    PGN_FUEL_CELL_COMPARTMENT_INFORMATION : UDINT := UDINT#16#F349; (* < 62281 - FCCI *)
    PGN_GENSET_REAL_POWER_SETPOINT_DEMAND : UDINT := UDINT#16#F34A; (* < 62282 - GRPSD *)
    PGN_GENSET_REAL_POWER_CONTROL_2 : UDINT := UDINT#16#F34B; (* < 62283 - GRPC2 *)
    PGN_HIGH_VOLTAGE_ENERGY_STORAGE_PACK_1_DATA_12 : UDINT := UDINT#16#F34C; (* < 62284 - HVESP1D12 *)
    PGN_HIGH_VOLTAGE_ENERGY_STORAGE_PACK_1_DATA_13 : UDINT := UDINT#16#F34D; (* < 62285 - HVESP1D13 *)
    PGN_HIGH_VOLTAGE_ENERGY_STORAGE_PACK_2_DATA_12 : UDINT := UDINT#16#F34E; (* < 62286 - HVESP2D12 *)
    PGN_HIGH_VOLTAGE_ENERGY_STORAGE_PACK_2_DATA_13 : UDINT := UDINT#16#F34F; (* < 62287 - HVESP2D13 *)
    PGN_HIGH_VOLTAGE_ENERGY_STORAGE_PACK_3_DATA_12 : UDINT := UDINT#16#F350; (* < 62288 - HVESP3D12 *)
    PGN_HIGH_VOLTAGE_ENERGY_STORAGE_PACK_3_DATA_13 : UDINT := UDINT#16#F351; (* < 62289 - HVESP3D13 *)
    PGN_HIGH_VOLTAGE_ENERGY_STORAGE_PACK_4_DATA_12 : UDINT := UDINT#16#F352; (* < 62290 - HVESP4D12 *)
    PGN_HIGH_VOLTAGE_ENERGY_STORAGE_PACK_4_DATA_13 : UDINT := UDINT#16#F353; (* < 62291 - HVESP4D13 *)
    PGN_HIGH_VOLTAGE_ENERGY_STORAGE_PACK_5_DATA_12 : UDINT := UDINT#16#F354; (* < 62292 - HVESP5D12 *)
    PGN_HIGH_VOLTAGE_ENERGY_STORAGE_PACK_5_DATA_13 : UDINT := UDINT#16#F355; (* < 62293 - HVESP5D13 *)
    PGN_HIGH_VOLTAGE_ENERGY_STORAGE_PACK_6_DATA_12 : UDINT := UDINT#16#F356; (* < 62294 - HVESP6D12 *)
    PGN_HIGH_VOLTAGE_ENERGY_STORAGE_PACK_6_DATA_13 : UDINT := UDINT#16#F357; (* < 62295 - HVESP6D13 *)
    PGN_HIGH_VOLTAGE_ENERGY_STORAGE_PACK_7_DATA_12 : UDINT := UDINT#16#F358; (* < 62296 - HVESP7D12 *)
    PGN_HIGH_VOLTAGE_ENERGY_STORAGE_PACK_7_DATA_13 : UDINT := UDINT#16#F359; (* < 62297 - HVESP7D13 *)
    PGN_HIGH_VOLTAGE_ENERGY_STORAGE_PACK_8_DATA_12 : UDINT := UDINT#16#F35A; (* < 62298 - HVESP8D12 *)
    PGN_HIGH_VOLTAGE_ENERGY_STORAGE_PACK_8_DATA_13 : UDINT := UDINT#16#F35B; (* < 62299 - HVESP8D13 *)
    PGN_HIGH_VOLTAGE_ENERGY_STORAGE_PACK_9_DATA_12 : UDINT := UDINT#16#F35C; (* < 62300 - HVESP9D12 *)
    PGN_HIGH_VOLTAGE_ENERGY_STORAGE_PACK_9_DATA_13 : UDINT := UDINT#16#F35D; (* < 62301 - HVESP9D13 *)
    PGN_HIGH_VOLTAGE_ENERGY_STORAGE_PACK_10_DATA_12 : UDINT := UDINT#16#F35E; (* < 62302 - HVESP10D12 *)
    PGN_HIGH_VOLTAGE_ENERGY_STORAGE_PACK_10_DATA_13 : UDINT := UDINT#16#F35F; (* < 62303 - HVESP10D13 *)
    PGN_HIGH_VOLTAGE_ENERGY_STORAGE_PACK_11_DATA_12 : UDINT := UDINT#16#F360; (* < 62304 - HVESP11D12 *)
    PGN_HIGH_VOLTAGE_ENERGY_STORAGE_PACK_11_DATA_13 : UDINT := UDINT#16#F361; (* < 62305 - HVESP11D13 *)
    PGN_HIGH_VOLTAGE_ENERGY_STORAGE_PACK_12_DATA_12 : UDINT := UDINT#16#F362; (* < 62306 - HVESP12D12 *)
    PGN_HIGH_VOLTAGE_ENERGY_STORAGE_PACK_12_DATA_13 : UDINT := UDINT#16#F363; (* < 62307 - HVESP12D13 *)
    PGN_TRACKED_VEHICLE_DATA : UDINT := UDINT#16#F364; (* < 62308 - TVD *)
    PGN_ELECTRIFIED_ACCESSORY_PROPULSION_MOTOR_COOLANT_FAN_3_STATUS_2 : UDINT := UDINT#16#F365; (* < 62309 - EAPMCF3S2 *)
    PGN_ELECTRIFIED_ACCESSORY_PROPULSION_MOTOR_COOLANT_FAN_2_STATUS_2 : UDINT := UDINT#16#F366; (* < 62310 - EAPMCF2S2 *)
    PGN_ELECTRIFIED_ACCESSORY_PROPULSION_MOTOR_COOLANT_FAN_1_STATUS_2 : UDINT := UDINT#16#F367; (* < 62311 - EAPMCF1S2 *)
    PGN_ELECTRIFIED_ACCESSORY_POWER_ELECTRONICS_COOLANT_FAN_3_STATUS_2 : UDINT := UDINT#16#F368; (* < 62312 - EAPECF3S2 *)
    PGN_ELECTRIFIED_ACCESSORY_POWER_ELECTRONICS_COOLANT_FAN_2_STATUS_2 : UDINT := UDINT#16#F369; (* < 62313 - EAPECF2S2 *)
    PGN_ELECTRIFIED_ACCESSORY_POWER_ELECTRONICS_COOLANT_FAN_1_STATUS_2 : UDINT := UDINT#16#F36A; (* < 62314 - EAPECF1S2 *)
    PGN_ELECTRIFIED_ACCESSORY_PROPULSION_MOTOR_OIL_PUMP_STATUS_2 : UDINT := UDINT#16#F36B; (* < 62315 - EAPMOPS2 *)
    PGN_ELECTRIFIED_ACCESSORY_PROPULSION_MOTOR_COOLANT_PUMP_STATUS_2 : UDINT := UDINT#16#F36C; (* < 62316 - EAPMCPS2 *)
    PGN_ELECTRIFIED_ACCESSORY_POWER_ELECTRONICS_COOLANT_PUMP_STATUS_2 : UDINT := UDINT#16#F36D; (* < 62317 - EAPECPS2 *)
    PGN_ELECTRIFIED_ACCESSORY_GENERATOR_COOLANT_PUMP_STATUS_2 : UDINT := UDINT#16#F36E; (* < 62318 - EAGCPS2 *)
    PGN_ELECTRIFIED_ACCESSORY_GENERATOR_COOLANT_FAN_STATUS_2 : UDINT := UDINT#16#F36F; (* < 62319 - EAGCFS2 *)
    PGN_ELECTRIFIED_ACCESSORY_MOTOR_STATUS_2 : UDINT := UDINT#16#F370; (* < 62320 - EAMS2 *)
    PGN_FUEL_CELL_SYSTEM_CONTROLLER_INFORMATION : UDINT := UDINT#16#F371; (* < 62321 - FCSCI *)
    PGN_FUEL_CELL_SYSTEM_MINIMUM_POWER_INFORMATION : UDINT := UDINT#16#F372; (* < 62322 - FCSMNPI *)
    PGN_FUEL_CELL_SYSTEM_MAXIMUM_POWER_INFORMATION : UDINT := UDINT#16#F373; (* < 62323 - FCSMXPI *)
    PGN_FUEL_CELL_SYSTEM_MINIMUM_CURRENT_INFORMATION : UDINT := UDINT#16#F374; (* < 62324 - FCSMNCI *)
    PGN_FUEL_CELL_SYSTEM_MAXIMUM_CURRENT_INFORMATION : UDINT := UDINT#16#F375; (* < 62325 - FCSMXCI *)
    PGN_HYDROGEN_STORAGE_SYSTEM_INFORMATION : UDINT := UDINT#16#F376; (* < 62326 - HSSI *)
    PGN_FUEL_CELL_SYSTEM_OPERATING_STATE : UDINT := UDINT#16#F377; (* < 62327 - FCSOS *)
    PGN_FUEL_CELL_SYSTEM_OPERATIONS_REQUEST : UDINT := UDINT#16#F378; (* < 62328 - FCSOR *)
    PGN_FUEL_CELL_STACK_INFORMATION : UDINT := UDINT#16#F379; (* < 62329 - FCSI *)
    PGN_FUEL_CELL_SYSTEM_COOLANT_FAN_1_STATUS_2 : UDINT := UDINT#16#F37A; (* < 62330 - FCSCF1S2 *)
    PGN_FUEL_CELL_SYSTEM_COOLANT_FAN_2_STATUS_2 : UDINT := UDINT#16#F37B; (* < 62331 - FCSCF2S2 *)
    PGN_FUEL_CELL_SYSTEM_COOLANT_FAN_3_STATUS_2 : UDINT := UDINT#16#F37C; (* < 62332 - FCSCF3S2 *)
    PGN_FUEL_CELL_SYSTEM_COOLANT_FAN_4_STATUS_2 : UDINT := UDINT#16#F37D; (* < 62333 - FCSCF4S2 *)
    PGN_HVESS_COOLANT_PUMP_1_STATUS_2 : UDINT := UDINT#16#F37E; (* < 62334 - HVESSCP1S2 *)
    PGN_HVESS_COOLANT_PUMP_2_STATUS_2 : UDINT := UDINT#16#F37F; (* < 62335 - HVESSCP2S2 *)
    PGN_HIGH_VOLTAGE_ENERGY_STORAGE_SYSTEM_FAN_STATUS_2 : UDINT := UDINT#16#F380; (* < 62336 - HVESSFS2 *)
    PGN_PTO_DRIVE_ENGAGEMENT_2 : UDINT := UDINT#16#F381; (* < 62337 - PTODE2 *)
    PGN_FUEL_CELL_SYSTEM_HYDROGEN_PRESSURE : UDINT := UDINT#16#F382; (* < 62338 - FCSHP *)
    PGN_ENGINE_GAS_FLOW_RATE_2 : UDINT := UDINT#16#F383; (* < 62339 - EGF2 *)
    PGN_ENGINE_SUPERCHARGER_INFORMATION : UDINT := UDINT#16#F384; (* < 62340 - ESI *)
    PGN_ENGINE_DISCONNECT_CLUTCH : UDINT := UDINT#16#F385; (* < 62341 - EDC *)
    PGN_GNSS_CORRECTION_DATA : UDINT := UDINT#16#F959; (* < 63833 - GNSSCD *)
    PGN_ENGINE_CRANKCASE_VENTILATION_HEATER_INFORMATION_3 : UDINT := UDINT#16#F95A; (* < 63834 - ECVHI3 *)
    PGN_ENGINE_CRANKCASE_VENTILATION_HEATER_INFORMATION_2 : UDINT := UDINT#16#F95B; (* < 63835 - ECVHI2 *)
    PGN_ENGINE_CRANKCASE_VENTILATION_HEATER_INFORMATION_1 : UDINT := UDINT#16#F95C; (* < 63836 - ECVHI1 *)
    PGN_AIR_FUEL_RATIO_2 : UDINT := UDINT#16#F95D; (* < 63837 - AFR2 *)
    PGN_OBFCM_ENGINE_OUTPUT_ENERGY_STATIC_DATA : UDINT := UDINT#16#F95E; (* < 63838 - OBFCME *)
    PGN_OBFCM_VEHICLE_DISTANCE_STATIC_DATA : UDINT := UDINT#16#F95F; (* < 63839 - OBFCMD *)
    PGN_OBFCM_FUEL_2_STATIC_DATA : UDINT := UDINT#16#F960; (* < 63840 - OBFCMF2 *)
    PGN_OBFCM_FUEL_1_STATIC_DATA : UDINT := UDINT#16#F961; (* < 63841 - OBFCMF1 *)
    PGN_OBFCM_COUNTERS : UDINT := UDINT#16#F962; (* < 63842 - OBFCMC *)
    PGN_OBFCM_ACCUMULATORS : UDINT := UDINT#16#F963; (* < 63843 - OBFCMA *)
    PGN_OBFCM_FUEL_CONSUMPTION : UDINT := UDINT#16#F964; (* < 63844 - OBFCMFC *)
    PGN_ENGINE_VVT_SYSTEM_DATA : UDINT := UDINT#16#F965; (* < 63845 - EVVT *)
    PGN_MAINTENANCE_INFORMATION_2 : UDINT := UDINT#16#F966; (* < 63846 - MI2 *)
    PGN_ALTERNATE_FUEL_7 : UDINT := UDINT#16#F967; (* < 63847 - AF7 *)
    PGN_ENGINE_CATALYST_DIVERTER_ACTUATOR_INFORMATION : UDINT := UDINT#16#F968; (* < 63848 - ECDAI *)
    PGN_ELECTRONIC_LOGGING_DEVICE_HOURS_OF_SERVICE : UDINT := UDINT#16#F969; (* < 63849 - ELDHOS *)
    PGN_ER_DC_DC_CONVERTER_4_REFERENCES : UDINT := UDINT#16#F96A; (* < 63850 - ERDCDC4RF *)
    PGN_ER_DC_DC_CONVERTER_4_POWER_LIMITS_REQUEST : UDINT := UDINT#16#F96B; (* < 63851 - ERDCDC4PLR *)
    PGN_ER_DC_DC_CONVERTER_4_CURRENT_LIMITS_REQUEST : UDINT := UDINT#16#F96C; (* < 63852 - ERDCDC4CLR *)
    PGN_ER_DC_DC_CONVERTER_4_VOLTAGE_LIMITS_REQUEST : UDINT := UDINT#16#F96D; (* < 63853 - ERDCDC4VLR *)
    PGN_ER_DC_DC_CONVERTER_4_TEMPERATURES : UDINT := UDINT#16#F96E; (* < 63854 - ERDCDC4T *)
    PGN_ER_DC_DC_CONVERTER_4_POWER_LIMIT_SETTINGS : UDINT := UDINT#16#F96F; (* < 63855 - ERDCDC4PLS *)
    PGN_ER_DC_DC_CONVERTER_4_CURRENT_LIMITS_SETTINGS : UDINT := UDINT#16#F970; (* < 63856 - ERDCDC4CLS *)
    PGN_ER_DC_DC_CONVERTER_4_VOLTAGE_LIMIT_SETTINGS : UDINT := UDINT#16#F971; (* < 63857 - ERDCDC4VLS *)
    PGN_ER_DC_DC_CONVERTER_4_LOW_VOLTAGE : UDINT := UDINT#16#F972; (* < 63858 - ERDCDC4LV *)
    PGN_ER_DC_DC_CONVERTER_4_POWER_AND_CHASSIS_VOLTAGE : UDINT := UDINT#16#F973; (* < 63859 - ERDCDC4PCV *)
    PGN_ER_DC_DC_CONVERTER_4_VOLTAGE_AND_CURRENT : UDINT := UDINT#16#F974; (* < 63860 - ERDCDC4VC *)
    PGN_ER_DC_DC_CONVERTER_4_OPERATING_STATUS : UDINT := UDINT#16#F975; (* < 63861 - ERDCDC4OS *)
    PGN_ER_DC_DC_CONVERTER_4_CONTROL : UDINT := UDINT#16#F976; (* < 63862 - ERDCDC4C *)
    PGN_ER_DC_DC_CONVERTER_3_REFERENCES : UDINT := UDINT#16#F977; (* < 63863 - ERDCDC3RF *)
    PGN_ER_DC_DC_CONVERTER_3_POWER_LIMITS_REQUEST : UDINT := UDINT#16#F978; (* < 63864 - ERDCDC3PLR *)
    PGN_ER_DC_DC_CONVERTER_3_CURRENT_LIMITS_REQUEST : UDINT := UDINT#16#F979; (* < 63865 - ERDCDC3CLR *)
    PGN_ER_DC_DC_CONVERTER_3_VOLTAGE_LIMITS_REQUEST : UDINT := UDINT#16#F97A; (* < 63866 - ERDCDC3VLR *)
    PGN_ER_DC_DC_CONVERTER_3_TEMPERATURES : UDINT := UDINT#16#F97B; (* < 63867 - ERDCDC3T *)
    PGN_ER_DC_DC_CONVERTER_3_POWER_LIMIT_SETTINGS : UDINT := UDINT#16#F97C; (* < 63868 - ERDCDC3PLS *)
    PGN_ER_DC_DC_CONVERTER_3_CURRENT_LIMITS_SETTINGS : UDINT := UDINT#16#F97D; (* < 63869 - ERDCDC3CLS *)
    PGN_ER_DC_DC_CONVERTER_3_VOLTAGE_LIMIT_SETTINGS : UDINT := UDINT#16#F97E; (* < 63870 - ERDCDC3VLS *)
    PGN_ER_DC_DC_CONVERTER_3_LOW_VOLTAGE : UDINT := UDINT#16#F97F; (* < 63871 - ERDCDC3LV *)
    PGN_ER_DC_DC_CONVERTER_3_POWER_AND_CHASSIS_VOLTAGE : UDINT := UDINT#16#F980; (* < 63872 - ERDCDC3PCV *)
    PGN_ER_DC_DC_CONVERTER_3_VOLTAGE_AND_CURRENT : UDINT := UDINT#16#F981; (* < 63873 - ERDCDC3VC *)
    PGN_ER_DC_DC_CONVERTER_3_OPERATING_STATUS : UDINT := UDINT#16#F982; (* < 63874 - ERDCDC3OS *)
    PGN_ER_DC_DC_CONVERTER_3_CONTROL : UDINT := UDINT#16#F983; (* < 63875 - ERDCDC3C *)
    PGN_ER_DC_DC_CONVERTER_2_REFERENCES : UDINT := UDINT#16#F984; (* < 63876 - ERDCDC2RF *)
    PGN_ER_DC_DC_CONVERTER_2_POWER_LIMITS_REQUEST : UDINT := UDINT#16#F985; (* < 63877 - ERDCDC2PLR *)
    PGN_ER_DC_DC_CONVERTER_2_CURRENT_LIMITS_REQUEST : UDINT := UDINT#16#F986; (* < 63878 - ERDCDC2CLR *)
    PGN_ER_DC_DC_CONVERTER_2_VOLTAGE_LIMITS_REQUEST : UDINT := UDINT#16#F987; (* < 63879 - ERDCDC2VLR *)
    PGN_ER_DC_DC_CONVERTER_2_TEMPERATURES : UDINT := UDINT#16#F988; (* < 63880 - ERDCDC2T *)
    PGN_ER_DC_DC_CONVERTER_2_POWER_LIMIT_SETTINGS : UDINT := UDINT#16#F989; (* < 63881 - ERDCDC2PLS *)
    PGN_ER_DC_DC_CONVERTER_2_CURRENT_LIMITS_SETTINGS : UDINT := UDINT#16#F98A; (* < 63882 - ERDCDC2CLS *)
    PGN_ER_DC_DC_CONVERTER_2_VOLTAGE_LIMIT_SETTINGS : UDINT := UDINT#16#F98B; (* < 63883 - ERDCDC2VLS *)
    PGN_ER_DC_DC_CONVERTER_2_LOW_VOLTAGE : UDINT := UDINT#16#F98C; (* < 63884 - ERDCDC2LV *)
    PGN_ER_DC_DC_CONVERTER_2_POWER_AND_CHASSIS_VOLTAGE : UDINT := UDINT#16#F98D; (* < 63885 - ERDCDC2PCV *)
    PGN_ER_DC_DC_CONVERTER_2_VOLTAGE_AND_CURRENT : UDINT := UDINT#16#F98E; (* < 63886 - ERDCDC2VC *)
    PGN_ER_DC_DC_CONVERTER_2_OPERATING_STATUS : UDINT := UDINT#16#F98F; (* < 63887 - ERDCDC2OS *)
    PGN_ER_DC_DC_CONVERTER_2_CONTROL : UDINT := UDINT#16#F990; (* < 63888 - ERDCDC2C *)
    PGN_ER_DC_DC_CONVERTER_1_REFERENCES : UDINT := UDINT#16#F991; (* < 63889 - ERDCDC1RF *)
    PGN_ER_DC_DC_CONVERTER_1_POWER_LIMITS_REQUEST : UDINT := UDINT#16#F992; (* < 63890 - ERDCDC1PLR *)
    PGN_ER_DC_DC_CONVERTER_1_CURRENT_LIMITS_REQUEST : UDINT := UDINT#16#F993; (* < 63891 - ERDCDC1CLR *)
    PGN_ER_DC_DC_CONVERTER_1_VOLTAGE_LIMITS_REQUEST : UDINT := UDINT#16#F994; (* < 63892 - ERDCDC1VLR *)
    PGN_ER_DC_DC_CONVERTER_1_TEMPERATURES : UDINT := UDINT#16#F995; (* < 63893 - ERDCDC1T *)
    PGN_ER_DC_DC_CONVERTER_1_POWER_LIMIT_SETTINGS : UDINT := UDINT#16#F996; (* < 63894 - ERDCDC1PLS *)
    PGN_ER_DC_DC_CONVERTER_1_CURRENT_LIMITS_SETTINGS : UDINT := UDINT#16#F997; (* < 63895 - ERDCDC1CLS *)
    PGN_ER_DC_DC_CONVERTER_1_VOLTAGE_LIMIT_SETTINGS : UDINT := UDINT#16#F998; (* < 63896 - ERDCDC1VLS *)
    PGN_ER_DC_DC_CONVERTER_1_LOW_VOLTAGE : UDINT := UDINT#16#F999; (* < 63897 - ERDCDC1LV *)
    PGN_ER_DC_DC_CONVERTER_1_POWER_AND_CHASSIS_VOLTAGE : UDINT := UDINT#16#F99A; (* < 63898 - ERDCDC1PCV *)
    PGN_ER_DC_DC_CONVERTER_1_VOLTAGE_AND_CURRENT : UDINT := UDINT#16#F99B; (* < 63899 - ERDCDC1VC *)
    PGN_ER_DC_DC_CONVERTER_1_OPERATING_STATUS : UDINT := UDINT#16#F99C; (* < 63900 - ERDCDC1OS *)
    PGN_ER_DC_DC_CONVERTER_1_CONTROL : UDINT := UDINT#16#F99D; (* < 63901 - ERDCDC1C *)
    PGN_CAB_AIR_QUALITY_SYSTEM_INFORMATION_2 : UDINT := UDINT#16#F99E; (* < 63902 - CAQSI2 *)
    PGN_CAB_AIR_QUALITY_SYSTEM_INFORMATION_1 : UDINT := UDINT#16#F99F; (* < 63903 - CAQSI1 *)
    PGN_WELL_STIMULATION_PUMP_SYSTEM_6 : UDINT := UDINT#16#F9A0; (* < 63904 - WSP6 *)
    PGN_ENGINE_FUEL_LUBE_SYSTEMS_4 : UDINT := UDINT#16#F9A1; (* < 63905 - EFS4 *)
    PGN_ALTERNATE_FUEL_6 : UDINT := UDINT#16#F9A2; (* < 63906 - AF6 *)
    PGN_ENGINE_CATALYST_DIVERTER_ACTUATOR_CONTROL : UDINT := UDINT#16#F9A3; (* < 63907 - ECDAC *)
    PGN_AMBIENT_CONDITIONS_4 : UDINT := UDINT#16#F9A4; (* < 63908 - AMB4 *)
    PGN_ENGINE_EXHAUST_PARTICULATE_CONTROL_SYSTEM_INFO_2 : UDINT := UDINT#16#F9A5; (* < 63909 - EEPCSI2 *)
    PGN_ENGINE_EXHAUST_PARTICULATE_CONTROL_SYSTEM_INFO_1 : UDINT := UDINT#16#F9A6; (* < 63910 - EEPCSI1 *)
    PGN_AFTERTREATMENT_SYSTEM_INFORMATION_20 : UDINT := UDINT#16#F9A7; (* < 63911 - ASI20 *)
    PGN_AFTERTREATMENT_SYSTEM_INFORMATION_19 : UDINT := UDINT#16#F9A8; (* < 63912 - ASI19 *)
    PGN_AFTERTREATMENT_SYSTEM_INFORMATION_18 : UDINT := UDINT#16#F9A9; (* < 63913 - ASI18 *)
    PGN_AFTERTREATMENT_SYSTEM_INFORMATION_17 : UDINT := UDINT#16#F9AA; (* < 63914 - ASI17 *)
    PGN_AFTERTREATMENT_SYSTEM_INFORMATION_16 : UDINT := UDINT#16#F9AB; (* < 63915 - ASI16 *)
    PGN_AFTERTREATMENT_SYSTEM_INFORMATION_15 : UDINT := UDINT#16#F9AC; (* < 63916 - ASI15 *)
    PGN_AFTERTREATMENT_SYSTEM_INFORMATION_14 : UDINT := UDINT#16#F9AD; (* < 63917 - ASI14 *)
    PGN_AFTERTREATMENT_SYSTEM_INFORMATION_13 : UDINT := UDINT#16#F9AE; (* < 63918 - ASI13 *)
    PGN_AFTERTREATMENT_SYSTEM_INFORMATION_12 : UDINT := UDINT#16#F9AF; (* < 63919 - ASI12 *)
    PGN_AFTERTREATMENT_SYSTEM_INFORMATION_11 : UDINT := UDINT#16#F9B0; (* < 63920 - ASI11 *)
    PGN_AFTERTREATMENT_SYSTEM_INFORMATION_10 : UDINT := UDINT#16#F9B1; (* < 63921 - ASI10 *)
    PGN_AFTERTREATMENT_SYSTEM_INFORMATION_9 : UDINT := UDINT#16#F9B2; (* < 63922 - ASI9 *)
    PGN_ROUTE_ATTRIBUTES_PROFILE : UDINT := UDINT#16#F9B3; (* < 63923 - RTAP *)
    PGN_GENSET_SUPPORTING_FUNCTIONS_2 : UDINT := UDINT#16#F9B4; (* < 63924 - GSF2 *)
    PGN_ALTERNATOR_INFORMATION_2 : UDINT := UDINT#16#F9B5; (* < 63925 - AS2 *)
    PGN_WELL_STIMULATION_PUMP_SYSTEM_5 : UDINT := UDINT#16#F9B6; (* < 63926 - WSP5 *)
    PGN_WELL_STIMULATION_PUMP_SYSTEM_4 : UDINT := UDINT#16#F9B7; (* < 63927 - WSP4 *)
    PGN_TIRE_INFORMATION : UDINT := UDINT#16#F9B8; (* < 63928 - TI *)
    PGN_HYDROGEN_SYSTEM_STATUS : UDINT := UDINT#16#F9B9; (* < 63929 - H2SS *)
    PGN_ROUTE_WAYPOINT_GPS_COORDINATES : UDINT := UDINT#16#F9BA; (* < 63930 - RWGPSC *)
    PGN_ROUTE_INFORMATION : UDINT := UDINT#16#F9BB; (* < 63931 - RTI *)
    PGN_ENGINE_FLUID_LEVEL_PRESSURE_15 : UDINT := UDINT#16#F9BC; (* < 63932 - EFL/P15 *)
    PGN_FUEL_CELL_SYSTEM_COOLANT_INFORMATION_3 : UDINT := UDINT#16#F9BD; (* < 63933 - FCSCI3 *)
    PGN_TRANSMISSION_CONFIGURATION_3 : UDINT := UDINT#16#F9BE; (* < 63934 - TCFG3 *)
    PGN_ENRICHMENT_INFORMATION : UDINT := UDINT#16#F9BF; (* < 63935 - ENRI *)
    PGN_FUEL_CELL_SYSTEM_VOLTAGE_LIMIT_COMMAND : UDINT := UDINT#16#F9C0; (* < 63936 - FCSVLC *)
    PGN_HYDROGEN_SYSTEM_INFORMATION : UDINT := UDINT#16#F9C2; (* < 63938 - H2SYSINF *)
    PGN_AUXILIARY_INPUT_OUTPUT_STATUS_17 : UDINT := UDINT#16#F9C3; (* < 63939 - AUXIO17 *)
    PGN_AUXILIARY_INPUT_OUTPUT_STATUS_16 : UDINT := UDINT#16#F9C4; (* < 63940 - AUXIO16 *)
    PGN_AUXILIARY_INPUT_OUTPUT_STATUS_15 : UDINT := UDINT#16#F9C5; (* < 63941 - AUXIO15 *)
    PGN_AUXILIARY_INPUT_OUTPUT_STATUS_14 : UDINT := UDINT#16#F9C6; (* < 63942 - AUXIO14 *)
    PGN_AUXILIARY_INPUT_OUTPUT_STATUS_13 : UDINT := UDINT#16#F9C7; (* < 63943 - AUXIO13 *)
    PGN_AUXILIARY_INPUT_OUTPUT_STATUS_12 : UDINT := UDINT#16#F9C8; (* < 63944 - AUXIO12 *)
    PGN_AUXILIARY_INPUT_OUTPUT_STATUS_11 : UDINT := UDINT#16#F9C9; (* < 63945 - AUXIO11 *)
    PGN_AUXILIARY_INPUT_OUTPUT_STATUS_10 : UDINT := UDINT#16#F9CA; (* < 63946 - AUXIO10 *)
    PGN_AUXILIARY_INPUT_OUTPUT_STATUS_9 : UDINT := UDINT#16#F9CB; (* < 63947 - AUXIO9 *)
    PGN_AUXILIARY_INPUT_OUTPUT_STATUS_8 : UDINT := UDINT#16#F9CC; (* < 63948 - AUXIO8 *)
    PGN_AFTERTREATMENT_SYSTEM_INFORMATION_8 : UDINT := UDINT#16#F9CD; (* < 63949 - ASI8 *)
    PGN_BRAKE_TEMPERATURE_6 : UDINT := UDINT#16#F9CE; (* < 63950 - BKT6 *)
    PGN_BRAKE_TEMPERATURE_5 : UDINT := UDINT#16#F9CF; (* < 63951 - BKT5 *)
    PGN_BRAKE_TEMPERATURE_4 : UDINT := UDINT#16#F9D0; (* < 63952 - BKT4 *)
    PGN_BRAKE_TEMPERATURE_3 : UDINT := UDINT#16#F9D1; (* < 63953 - BKT3 *)
    PGN_BRAKE_TEMPERATURE_2 : UDINT := UDINT#16#F9D2; (* < 63954 - BKT2 *)
    PGN_BRAKE_TEMPERATURE_1 : UDINT := UDINT#16#F9D3; (* < 63955 - BKT1 *)
    PGN_WHEEL_BRAKE_LINING_REMAINING_INFORMATION_3 : UDINT := UDINT#16#F9D4; (* < 63956 - EBC7 *)
    PGN_WHEEL_BRAKE_LINING_REMAINING_INFORMATION_2 : UDINT := UDINT#16#F9D5; (* < 63957 - EBC6 *)
    PGN_HIGH_VOLTAGE_BUS_CONTACTOR_STATUS_3 : UDINT := UDINT#16#F9D6; (* < 63958 - HVBCS3 *)
    PGN_HIGH_VOLTAGE_BUS_CONTACTOR_STATUS_2 : UDINT := UDINT#16#F9D7; (* < 63959 - HVBCS2 *)
    PGN_HIGH_VOLTAGE_BUS_CONNECTION_COMMAND_2 : UDINT := UDINT#16#F9D8; (* < 63960 - HVBCC2 *)
    PGN_CAB_ILLUMINATION_DATA : UDINT := UDINT#16#F9D9; (* < 63961 - CID *)
    PGN_SERVICE_NEEDED_DTC_INFORMATION : UDINT := UDINT#16#F9DA; (* < 63962 - SNDI *)
    PGN_EVSE_STATUS_2 : UDINT := UDINT#16#F9DB; (* < 63963 - EVSES2 *)
    PGN_HIGH_VOLTAGE_ENERGY_STORAGE_SYSTEM_THERMAL_MANAGEMENT_SYSTEM_CHILLER_1 : UDINT := UDINT#16#F9DC; (* < 63964 - HVESSTCH1 *)
    PGN_HIGH_VOLTAGE_ENERGY_STORAGE_SYSTEM_THERMAL_MANAGEMENT_SYSTEM_CHILLER_2 : UDINT := UDINT#16#F9DD; (* < 63965 - HVESSTCH2 *)
    PGN_HIGH_VOLTAGE_ENERGY_STORAGE_SYSTEM_THERMAL_MANAGEMENT_SYSTEM_CHILLER_3 : UDINT := UDINT#16#F9DE; (* < 63966 - HVESSTCH3 *)
    PGN_HVESS_COOLANT_PUMP_1_STATUS_1 : UDINT := UDINT#16#F9DF; (* < 63967 - HVESSCP1S1 *)
    PGN_HVESS_COOLANT_PUMP_1_COMMAND : UDINT := UDINT#16#F9E0; (* < 63968 - HVESSCP1C *)
    PGN_HVESS_COOLANT_PUMP_2_STATUS_1 : UDINT := UDINT#16#F9E1; (* < 63969 - HVESSCP2S1 *)
    PGN_HVESS_COOLANT_PUMP_2_COMMAND : UDINT := UDINT#16#F9E2; (* < 63970 - HVESSCP2C *)
    PGN_HYDROGEN_SENSOR_INFORMATION : UDINT := UDINT#16#F9E3; (* < 63971 - H2SNSINF *)
    PGN_OPERATOR_INDUCEMENT_INFORMATION_2 : UDINT := UDINT#16#F9E4; (* < 63972 - OII2 *)
    PGN_OPERATOR_INDUCEMENT_VEHICLE_SPEED_INFORMATION_1 : UDINT := UDINT#16#F9E5; (* < 63973 - OIVSI1 *)
    PGN_OPERATOR_INDUCEMENT_VEHICLE_SPEED_INFORMATION_2 : UDINT := UDINT#16#F9E6; (* < 63974 - OIVSI2 *)
    PGN_ENGINE_PROTECTION_SPEED_DERATE_INFORMATION : UDINT := UDINT#16#F9E7; (* < 63975 - EPSDI *)
    PGN_ENGINE_PROTECTION_TORQUE_DERATE_INFORMATION : UDINT := UDINT#16#F9E8; (* < 63976 - EPTDI *)
    PGN_AFTERTREATMENT_SYSTEM_INFORMATION_7 : UDINT := UDINT#16#F9E9; (* < 63977 - ASI7 *)
    PGN_SAE_J2012_3_BYTE_DTC_DISPLAY : UDINT := UDINT#16#F9EA; (* < 63978 - J2012_3B *)
    PGN_HIGH_VOLTAGE_ENERGY_STORAGE_SYSTEM_INTERNAL_STATUS_5 : UDINT := UDINT#16#F9EB; (* < 63979 - HVESSIS5 *)
    PGN_HIGH_VOLTAGE_ENERGY_STORAGE_SYSTEM_INTERNAL_STATUS_6 : UDINT := UDINT#16#F9EC; (* < 63980 - HVESSIS6 *)
    PGN_HIGH_VOLTAGE_ENERGY_STORAGE_SYSTEM_INTERNAL_STATUS_7 : UDINT := UDINT#16#F9ED; (* < 63981 - HVESSIS7 *)
    PGN_ENGINE_CYLINDER_AVERAGE_IGNITION_DELAY_ANGLE_1 : UDINT := UDINT#16#F9EE; (* < 63982 - ECAIDA1 *)
    PGN_ENGINE_CYLINDER_AVERAGE_IGNITION_DELAY_ANGLE_2 : UDINT := UDINT#16#F9EF; (* < 63983 - ECAIDA2 *)
    PGN_ENGINE_CYLINDER_AVERAGE_IGNITION_DELAY_ANGLE_3 : UDINT := UDINT#16#F9F0; (* < 63984 - ECAIDA3 *)
    PGN_ENGINE_CYLINDER_AVERAGE_IGNITION_DELAY_ANGLE_4 : UDINT := UDINT#16#F9F1; (* < 63985 - ECAIDA4 *)
    PGN_ENGINE_CYLINDER_AVERAGE_IGNITION_DELAY_ANGLE_5 : UDINT := UDINT#16#F9F2; (* < 63986 - ECAIDA5 *)
    PGN_ENGINE_INDICATED_MEAN_EFFECTIVE_PRESSURE_INFORMATION_1 : UDINT := UDINT#16#F9F3; (* < 63987 - EIMEPI1 *)
    PGN_ENGINE_INDICATED_MEAN_EFFECTIVE_PRESSURE_INFORMATION_2 : UDINT := UDINT#16#F9F4; (* < 63988 - EIMEPI2 *)
    PGN_ENGINE_INDICATED_MEAN_EFFECTIVE_PRESSURE_INFORMATION_3 : UDINT := UDINT#16#F9F5; (* < 63989 - EIMEPI3 *)
    PGN_FUEL_CELL_SYSTEM_COOLANT_FAN_1_COMMAND : UDINT := UDINT#16#F9F6; (* < 63990 - FCSCF1C *)
    PGN_FUEL_CELL_SYSTEM_COOLANT_FAN_1_STATUS_1 : UDINT := UDINT#16#F9F7; (* < 63991 - FCSCF1S1 *)
    PGN_FUEL_CELL_SYSTEM_COOLANT_FAN_2_COMMAND : UDINT := UDINT#16#F9F8; (* < 63992 - FCSCF2C *)
    PGN_FUEL_CELL_SYSTEM_COOLANT_FAN_2_STATUS_1 : UDINT := UDINT#16#F9F9; (* < 63993 - FCSCF2S1 *)
    PGN_FUEL_CELL_SYSTEM_COOLANT_FAN_3_COMMAND : UDINT := UDINT#16#F9FA; (* < 63994 - FCSCF3C *)
    PGN_FUEL_CELL_SYSTEM_COOLANT_FAN_3_STATUS_1 : UDINT := UDINT#16#F9FB; (* < 63995 - FCSCF3S1 *)
    PGN_FUEL_CELL_SYSTEM_COOLANT_FAN_4_COMMAND : UDINT := UDINT#16#F9FC; (* < 63996 - FCSCF4C *)
    PGN_FUEL_CELL_SYSTEM_COOLANT_FAN_4_STATUS_1 : UDINT := UDINT#16#F9FD; (* < 63997 - FCSCF4S1 *)
    PGN_APIS_SUPPORTED : UDINT := UDINT#16#F9FE; (* < 63998 - APISUP *)
    PGN_FUEL_CELL_SYSTEM_CONFIGURATION : UDINT := UDINT#16#F9FF; (* < 63999 - FCSC *)
    PGN_FUEL_CELL_SYSTEM_COOLANT_INFORMATION_1 : UDINT := UDINT#16#FA00; (* < 64000 - FCSCI1 *)
    PGN_FUEL_CELL_SYSTEM_COOLANT_INFORMATION_2 : UDINT := UDINT#16#FA01; (* < 64001 - FCSCI2 *)
    PGN_DASH_DISPLAY_3 : UDINT := UDINT#16#FA06; (* < 64006 - DD3 *)
    PGN_VEHICLE_SPEED_PROFILE : UDINT := UDINT#16#FA07; (* < 64007 - VSP *)
    PGN_REFERENCE_TIME : UDINT := UDINT#16#FA08; (* < 64008 - REFTIME *)
    PGN_SOFTWARE_HISTORY : UDINT := UDINT#16#FA09; (* < 64009 - SH *)
    PGN_MOTOR_GENERATOR_1_THERMAL_PERFORMANCE_STATUS : UDINT := UDINT#16#FA0A; (* < 64010 - MG1TPS *)
    PGN_MOTOR_GENERATOR_2_THERMAL_PERFORMANCE_STATUS : UDINT := UDINT#16#FA0B; (* < 64011 - MG2TPS *)
    PGN_MOTOR_GENERATOR_3_THERMAL_PERFORMANCE_STATUS : UDINT := UDINT#16#FA0C; (* < 64012 - MG3TPS *)
    PGN_MOTOR_GENERATOR_4_THERMAL_PERFORMANCE_STATUS : UDINT := UDINT#16#FA0D; (* < 64013 - MG4TPS *)
    PGN_MOTOR_GENERATOR_5_THERMAL_PERFORMANCE_STATUS : UDINT := UDINT#16#FA0E; (* < 64014 - MG5TPS *)
    PGN_MOTOR_GENERATOR_6_THERMAL_PERFORMANCE_STATUS : UDINT := UDINT#16#FA0F; (* < 64015 - MG6TPS *)
    PGN_ON_BOARD_PROGRAMMING_EVENT_TIME_DATE : UDINT := UDINT#16#FA10; (* < 64016 - OBPETD *)
    PGN_AFTERTREATMENT_1_LIGHT_OFF_SCR_SERVICE_INFORMATION_1 : UDINT := UDINT#16#FA11; (* < 64017 - A1LOSCRSI1 *)
    PGN_MOTOR_GENERATOR_LOCATION_EXTENDED : UDINT := UDINT#16#FA12; (* < 64018 - MGLE *)
    PGN_COLD_START_EMISSIONS_REDUCTION_STRATEGY_CURRENT_OPERATING_CYCLE_DATA : UDINT := UDINT#16#FA13; (* < 64019 - CSERSC *)
    PGN_COLD_START_EMISSIONS_REDUCTION_STRATEGY_AVERAGE_DATA : UDINT := UDINT#16#FA14; (* < 64020 - CSERSA *)
    PGN_GENSET_SUPPORTING_FUNCTIONS : UDINT := UDINT#16#FA15; (* < 64021 - GSF *)
    PGN_HIGH_VOLTAGE_ENERGY_STORAGE_SYSTEM_INTERNAL_STATUS_1 : UDINT := UDINT#16#FA16; (* < 64022 - HVESSIS1 *)
    PGN_HIGH_VOLTAGE_ENERGY_STORAGE_SYSTEM_INTERNAL_STATUS_2 : UDINT := UDINT#16#FA17; (* < 64023 - HVESSIS2 *)
    PGN_HIGH_VOLTAGE_ENERGY_STORAGE_SYSTEM_INTERNAL_STATUS_3 : UDINT := UDINT#16#FA18; (* < 64024 - HVESSIS3 *)
    PGN_HIGH_VOLTAGE_ENERGY_STORAGE_SYSTEM_INTERNAL_STATUS_4 : UDINT := UDINT#16#FA19; (* < 64025 - HVESSIS4 *)
    PGN_ELECTRONIC_ENGINE_CONTROLLER_23 : UDINT := UDINT#16#FA1A; (* < 64026 - EEC23 *)
    PGN_ELECTRONIC_ENGINE_CONTROLLER_24 : UDINT := UDINT#16#FA1B; (* < 64027 - EEC24 *)
    PGN_ELECTRONIC_ENGINE_CONTROLLER_25 : UDINT := UDINT#16#FA1C; (* < 64028 - EEC25 *)
    PGN_HIGH_VOLTAGE_BUS_CONNECTION_COMMAND_1 : UDINT := UDINT#16#FA1D; (* < 64029 - HVBCC1 *)
    PGN_HIGH_VOLTAGE_BUS_CONTACTOR_STATUS_1 : UDINT := UDINT#16#FA1E; (* < 64030 - HVBCS1 *)
    PGN_AFTERTREATMENT_SYSTEM_INFORMATION_6 : UDINT := UDINT#16#FA1F; (* < 64031 - ASI6 *)
    PGN_EV_MULTI_CONNECTION_DC_CHARGING_LIMITS_2 : UDINT := UDINT#16#FA20; (* < 64032 - EVMCDCLIM2 *)
    PGN_EV_MULTI_CONNECTION_CHARGING_IN_PROGRESS : UDINT := UDINT#16#FA21; (* < 64033 - EVMCDCCIP *)
    PGN_SENSOR_SUPPLY_VOLTAGE : UDINT := UDINT#16#FA22; (* < 64034 - SSV *)
    PGN_MOTOR_GENERATOR_LOCATION_OBSOLETE_USE_PGN_64018 : UDINT := UDINT#16#FA23; (* < 64035 - MGL *)
    PGN_HIGH_VOLTAGE_ENERGY_STORAGE_SYSTEM_DATA_12 : UDINT := UDINT#16#FA24; (* < 64036 - HVESSD12 *)
    PGN_HIGH_VOLTAGE_ENERGY_STORAGE_SYSTEM_DATA_13 : UDINT := UDINT#16#FA25; (* < 64037 - HVESSD13 *)
    PGN_HIGH_VOLTAGE_ENERGY_STORAGE_SYSTEM_DATA_14 : UDINT := UDINT#16#FA26; (* < 64038 - HVESSD14 *)
    PGN_HIGH_VOLTAGE_ENERGY_STORAGE_PACK_1_INTERNAL_STATUS_1 : UDINT := UDINT#16#FA27; (* < 64039 - HVESP1IS1 *)
    PGN_HIGH_VOLTAGE_ENERGY_STORAGE_PACK_2_INTERNAL_STATUS_1 : UDINT := UDINT#16#FA28; (* < 64040 - HVESP2IS1 *)
    PGN_HIGH_VOLTAGE_ENERGY_STORAGE_PACK_3_INTERNAL_STATUS_1 : UDINT := UDINT#16#FA29; (* < 64041 - HVESP3IS1 *)
    PGN_HIGH_VOLTAGE_ENERGY_STORAGE_PACK_4_INTERNAL_STATUS_1 : UDINT := UDINT#16#FA2A; (* < 64042 - HVESP4IS1 *)
    PGN_HIGH_VOLTAGE_ENERGY_STORAGE_PACK_5_INTERNAL_STATUS_1 : UDINT := UDINT#16#FA2B; (* < 64043 - HVESP5IS1 *)
    PGN_HIGH_VOLTAGE_ENERGY_STORAGE_PACK_6_INTERNAL_STATUS_1 : UDINT := UDINT#16#FA2C; (* < 64044 - HVESP6IS1 *)
    PGN_HIGH_VOLTAGE_ENERGY_STORAGE_PACK_7_INTERNAL_STATUS_1 : UDINT := UDINT#16#FA2D; (* < 64045 - HVESP7IS1 *)
    PGN_HIGH_VOLTAGE_ENERGY_STORAGE_PACK_8_INTERNAL_STATUS_1 : UDINT := UDINT#16#FA2E; (* < 64046 - HVESP8IS1 *)
    PGN_HIGH_VOLTAGE_ENERGY_STORAGE_PACK_9_INTERNAL_STATUS_1 : UDINT := UDINT#16#FA2F; (* < 64047 - HVESP9IS1 *)
    PGN_HIGH_VOLTAGE_ENERGY_STORAGE_PACK_10_INTERNAL_STATUS_1 : UDINT := UDINT#16#FA30; (* < 64048 - HVESP10IS1 *)
    PGN_HIGH_VOLTAGE_ENERGY_STORAGE_PACK_11_INTERNAL_STATUS_1 : UDINT := UDINT#16#FA31; (* < 64049 - HVESP11IS1 *)
    PGN_HIGH_VOLTAGE_ENERGY_STORAGE_PACK_12_INTERNAL_STATUS_1 : UDINT := UDINT#16#FA32; (* < 64050 - HVESP12IS1 *)
    PGN_MULTI_COLOR_INDICATOR_LAMP_COMMAND : UDINT := UDINT#16#FA33; (* < 64051 - MCILC *)
    PGN_MULTI_COLOR_INDICATOR_LAMP_STATUS : UDINT := UDINT#16#FA34; (* < 64052 - MCILS *)
    PGN_REFUSE_TRUCK_BODY_INFORMATION : UDINT := UDINT#16#FA35; (* < 64053 - RTBI *)
    PGN_ENGINE_FLUID_LEVEL_PRESSURE_14 : UDINT := UDINT#16#FA36; (* < 64054 - EFL/P14 *)
    PGN_WELL_STIMULATION_TRANSMISSION_CONTROL : UDINT := UDINT#16#FA37; (* < 64055 - WSTC *)
    PGN_WELL_STIMULATION_PUMP_PROTECTION_SYSTEM_CONFIGURATION_COMMAND_1 : UDINT := UDINT#16#FA38; (* < 64056 - WSPPS1 *)
    PGN_WELL_STIMULATION_PUMP_PROTECTION_SYSTEM_CONFIGURATION_COMMAND_2 : UDINT := UDINT#16#FA39; (* < 64057 - WSPPS2 *)
    PGN_ELECTRIC_PTO_DRIVE_ENGAGEMENT_1 : UDINT := UDINT#16#FA3A; (* < 64058 - EPTODE1 *)
    PGN_ELECTRIC_PTO_1_INFORMATION : UDINT := UDINT#16#FA3B; (* < 64059 - EPTO1I *)
    PGN_ENGINE_EXHAUST_O2_SENSOR_INFORMATION : UDINT := UDINT#16#FA3C; (* < 64060 - E02SI *)
    PGN_GASEOUS_FUEL_SUPPLY_PRESSURE_3 : UDINT := UDINT#16#FA3D; (* < 64061 - GFSP3 *)
    PGN_TRAFFIC_SIGNAGE : UDINT := UDINT#16#FA3E; (* < 64062 - TS *)
    PGN_ENGINE_CONFIGURATION_4 : UDINT := UDINT#16#FA3F; (* < 64063 - EC4 *)
    PGN_ELECTRONIC_TRANSMISSION_CONTROLLER_15 : UDINT := UDINT#16#FA40; (* < 64064 - ETC15 *)
    PGN_AUTOMATED_DRIVING_SYSTEM_NETWORK_CONFIGURATION_2 : UDINT := UDINT#16#FA41; (* < 64065 - ADSNC2 *)
    PGN_AUTOMATED_DRIVING_SYSTEM_NETWORK_CONFIGURATION_1 : UDINT := UDINT#16#FA42; (* < 64066 - ADSNC1 *)
    PGN_HYBRID_OR_EV_SYSTEM_INPUTS_2 : UDINT := UDINT#16#FA43; (* < 64067 - HSI2 *)
    PGN_ENGINE_SPEED_LOAD_FACTOR_INFORMATION_2 : UDINT := UDINT#16#FA44; (* < 64068 - LF2 *)
    PGN_GENERATOR_TRIP_ENERGY_2 : UDINT := UDINT#16#FA45; (* < 64069 - GTRACE2 *)
    PGN_SECURITY_SYSTEM_MACHINE_OPERATION_INFORMATION : UDINT := UDINT#16#FA46; (* < 64070 - SSMOI *)
    PGN_ENGINE_FUEL_ACTUATOR_SERVICE_MODE : UDINT := UDINT#16#FA47; (* < 64071 - EFASM *)
    PGN_STEERING_WHEEL_CONTROLS : UDINT := UDINT#16#FA48; (* < 64072 - STWCTRL *)
    PGN_PARK_ASSIST : UDINT := UDINT#16#FA49; (* < 64073 - PA *)
    PGN_EXTENDED_DTC_INFORMATION : UDINT := UDINT#16#FA4A; (* < 64074 - DM60 *)
    PGN_AFTERTREATMENT_2_SCR_DOSING_SYSTEM_INFORMATION_5 : UDINT := UDINT#16#FA4B; (* < 64075 - A2SCRDSI5 *)
    PGN_AFTERTREATMENT_1_SCR_DOSING_SYSTEM_INFORMATION_5 : UDINT := UDINT#16#FA4C; (* < 64076 - A1SCRDSI5 *)
    PGN_EV_ECONOMY_INFORMATION : UDINT := UDINT#16#FA4D; (* < 64077 - EVEI *)
    PGN_AUTOMATED_DRIVING_SYSTEM_STATUS_2 : UDINT := UDINT#16#FA4E; (* < 64078 - ADSS2 *)
    PGN_AUTOMATED_DRIVING_SYSTEM_CONTROL_3 : UDINT := UDINT#16#FA4F; (* < 64079 - ADSC3 *)
    PGN_AFTERCOOLER_VALVE : UDINT := UDINT#16#FA50; (* < 64080 - AV *)
    PGN_ENGINE_RADIATOR_1 : UDINT := UDINT#16#FA51; (* < 64081 - ER1 *)
    PGN_ENGINE_RADIATOR_2 : UDINT := UDINT#16#FA52; (* < 64082 - ER2 *)
    PGN_GENSET_ENCLOSURE_VENTILATION : UDINT := UDINT#16#FA53; (* < 64083 - GEV *)
    PGN_HEAT_EXCHANGER_1 : UDINT := UDINT#16#FA54; (* < 64084 - HE1 *)
    PGN_HEAT_EXCHANGER_2 : UDINT := UDINT#16#FA55; (* < 64085 - HE2 *)
    PGN_HEAT_EXCHANGER_3 : UDINT := UDINT#16#FA56; (* < 64086 - HE3 *)
    PGN_HEAT_EXCHANGER_4 : UDINT := UDINT#16#FA57; (* < 64087 - HE4 *)
    PGN_ENGINE_EXHAUST_GAS_HEAT_EXCHANGER : UDINT := UDINT#16#FA58; (* < 64088 - EEGHE *)
    PGN_GENSET_ENCLOSURE_VENTILATION_LOUVER : UDINT := UDINT#16#FA59; (* < 64089 - GEVL *)
    PGN_GENSET_EXTERNAL_COOLANT_SYSTEM : UDINT := UDINT#16#FA5A; (* < 64090 - GECS *)
    PGN_EV_DC_STATUS_1 : UDINT := UDINT#16#FA5B; (* < 64091 - EVDCS1 *)
    PGN_EVSE_DC_CHARGING_LIMITS_3 : UDINT := UDINT#16#FA5C; (* < 64092 - EVSEDCLIM3 *)
    PGN_EVSE_POWER_MAX_SCHEDULE : UDINT := UDINT#16#FA5D; (* < 64093 - EVSESCHED *)
    PGN_EV_CHARGE_PROFILE : UDINT := UDINT#16#FA5E; (* < 64094 - EVCHGPROF *)
    PGN_EV_DC_CHARGING_LIMITS_2 : UDINT := UDINT#16#FA5F; (* < 64095 - EVDCLIM2 *)
    PGN_EV_DC_CHARGING_IN_PROGRESS : UDINT := UDINT#16#FA60; (* < 64096 - EVDCCIP *)
    PGN_LIGHTING_DATA_2 : UDINT := UDINT#16#FA62; (* < 64098 - LD2 *)
    PGN_LIGHTING_COMMAND_2 : UDINT := UDINT#16#FA63; (* < 64099 - LCMD2 *)
    PGN_AFTERTREATMENT_SYSTEM_INFORMATION_5 : UDINT := UDINT#16#FA64; (* < 64100 - ASI5 *)
    PGN_AFTERTREATMENT_SYSTEM_INFORMATION_4 : UDINT := UDINT#16#FA65; (* < 64101 - ASI4 *)
    PGN_AFTERTREATMENT_SYSTEM_INFORMATION_3 : UDINT := UDINT#16#FA66; (* < 64102 - ASI3 *)
    PGN_FLUID_RESISTANCE_1 : UDINT := UDINT#16#FA67; (* < 64103 - FR1 *)
    PGN_POWER_CONVERTER_2_ISOLATION_INTEGRITY_REQUEST : UDINT := UDINT#16#FA68; (* < 64104 - PC2IIR *)
    PGN_POWER_CONVERTER_1_ISOLATION_INTEGRITY_REQUEST : UDINT := UDINT#16#FA69; (* < 64105 - PC1IIR *)
    PGN_POWER_CONVERTER_2_LIMITS_REQUEST_POWER : UDINT := UDINT#16#FA6A; (* < 64106 - PC2IRP *)
    PGN_POWER_CONVERTER_2_LIMITS_REQUEST_ELECTRICAL : UDINT := UDINT#16#FA6B; (* < 64107 - PC2ILRM *)
    PGN_POWER_CONVERTER_2_LIMITS_REQUEST_DC_ENERGY_SOURCE_1 : UDINT := UDINT#16#FA6C; (* < 64108 - PC2ILRDC *)
    PGN_POWER_CONVERTER_1_LIMITS_REQUEST_DC_ENERGY_SOURCE_1 : UDINT := UDINT#16#FA6D; (* < 64109 - PC1ILRDC *)
    PGN_POWER_CONVERTER_1_LIMITS_REQUEST_ELECTRICAL : UDINT := UDINT#16#FA6E; (* < 64110 - PC1ILRM *)
    PGN_POWER_CONVERTER_1_LIMITS_REQUEST_POWER : UDINT := UDINT#16#FA6F; (* < 64111 - PC1IRP *)
    PGN_INVERTER_1_LIFETIME_DATA : UDINT := UDINT#16#FA70; (* < 64112 - PC1LD *)
    PGN_INVERTER_2_LIFETIME_DATA : UDINT := UDINT#16#FA71; (* < 64113 - PC2LD *)
    PGN_POWER_CONVERTER_2_ACTIVE_POWER_LIMITS : UDINT := UDINT#16#FA72; (* < 64114 - PC2IAPL *)
    PGN_POWER_CONVERTER_1_ACTIVE_POWER_LIMITS : UDINT := UDINT#16#FA73; (* < 64115 - PC1IAPL *)
    PGN_POWER_CONVERTER_2_REFERENCE_1 : UDINT := UDINT#16#FA74; (* < 64116 - PC2IR1 *)
    PGN_POWER_CONVERTER_2_REFERENCE_2 : UDINT := UDINT#16#FA75; (* < 64117 - PC2IR2 *)
    PGN_POWER_CONVERTER_2_TEMPERATURE : UDINT := UDINT#16#FA76; (* < 64118 - PC2IT *)
    PGN_POWER_CONVERTER_1_TEMPERATURE : UDINT := UDINT#16#FA77; (* < 64119 - PC1IT *)
    PGN_POWER_CONVERTER_1_REFERENCE_2 : UDINT := UDINT#16#FA78; (* < 64120 - PC1IR2 *)
    PGN_POWER_CONVERTER_1_REFERENCE_1 : UDINT := UDINT#16#FA79; (* < 64121 - PC1IR1 *)
    PGN_POWER_CONVERTER_1_PHASE_CURRENT : UDINT := UDINT#16#FA7A; (* < 64122 - PC1PC *)
    PGN_POWER_CONVERTER_2_PHASE_CURRENT : UDINT := UDINT#16#FA7B; (* < 64123 - S21PC *)
    PGN_POWER_CONVERTER_1_PHASE_VOLTAGE : UDINT := UDINT#16#FA7C; (* < 64124 - PC1PV *)
    PGN_POWER_CONVERTER_2_PHASE_VOLTAGE : UDINT := UDINT#16#FA7D; (* < 64125 - PC2PV *)
    PGN_POWER_CONVERTER_POWER_MODULE_SWITCH_TEMPERATURES : UDINT := UDINT#16#FA7E; (* < 64126 - SIPST *)
    PGN_POWER_CONVERTER_1_POWER_MODULE_SWITCH_POWER_SUPPLY_VOLTAGE : UDINT := UDINT#16#FA7F; (* < 64127 - PC1PSV *)
    PGN_POWER_CONVERTER_2_POWER_MODULE_SWITCH_POWER_SUPPLY_VOLTAGE : UDINT := UDINT#16#FA80; (* < 64128 - PC2PSV *)
    PGN_POWER_CONVERTER_TOTALS_1 : UDINT := UDINT#16#FA81; (* < 64129 - SIT1 *)
    PGN_TRANSFORMER_TEMPERATURES : UDINT := UDINT#16#FA82; (* < 64130 - TFMRT *)
    PGN_ELECTRIFIED_ACCESSORY_ENGINE_COOLANT_PUMP_STATUS : UDINT := UDINT#16#FA83; (* < 64131 - EAECPS *)
    PGN_HIGH_VOLTAGE_ENERGY_STORAGE_PACK_11_HISTORY : UDINT := UDINT#16#FA84; (* < 64132 - HVESP11HIST *)
    PGN_HIGH_VOLTAGE_ENERGY_STORAGE_PACK_11_CONFIGURATION : UDINT := UDINT#16#FA85; (* < 64133 - HVESP11CFG *)
    PGN_HIGH_VOLTAGE_ENERGY_STORAGE_PACK_12_HISTORY : UDINT := UDINT#16#FA86; (* < 64134 - HVESP12HIST *)
    PGN_HIGH_VOLTAGE_ENERGY_STORAGE_PACK_12_CONFIGURATION : UDINT := UDINT#16#FA87; (* < 64135 - HVESP12CFG *)
    PGN_HIGH_VOLTAGE_ENERGY_STORAGE_PACK_13_HISTORY : UDINT := UDINT#16#FA88; (* < 64136 - HVESP13HIST *)
    PGN_HIGH_VOLTAGE_ENERGY_STORAGE_PACK_13_CONFIGURATION : UDINT := UDINT#16#FA89; (* < 64137 - HVESP13CFG *)
    PGN_HIGH_VOLTAGE_ENERGY_STORAGE_PACK_14_HISTORY : UDINT := UDINT#16#FA8A; (* < 64138 - HVESP14HIST *)
    PGN_HIGH_VOLTAGE_ENERGY_STORAGE_PACK_14_CONFIGURATION : UDINT := UDINT#16#FA8B; (* < 64139 - HVESP14CFG *)
    PGN_HIGH_VOLTAGE_ENERGY_STORAGE_PACK_15_HISTORY : UDINT := UDINT#16#FA8C; (* < 64140 - HVESP15HIST *)
    PGN_HIGH_VOLTAGE_ENERGY_STORAGE_PACK_15_CONFIGURATION : UDINT := UDINT#16#FA8D; (* < 64141 - HVESP15CFG *)
    PGN_HIGH_VOLTAGE_ENERGY_STORAGE_PACK_16_HISTORY : UDINT := UDINT#16#FA8E; (* < 64142 - HVESP16HIST *)
    PGN_HIGH_VOLTAGE_ENERGY_STORAGE_PACK_16_CONFIGURATION : UDINT := UDINT#16#FA8F; (* < 64143 - HVESP16CFG *)
    PGN_HIGH_VOLTAGE_ENERGY_STORAGE_PACK_17_HISTORY : UDINT := UDINT#16#FA90; (* < 64144 - HVESP17HIST *)
    PGN_HIGH_VOLTAGE_ENERGY_STORAGE_PACK_17_CONFIGURATION : UDINT := UDINT#16#FA91; (* < 64145 - HVESP17CFG *)
    PGN_HIGH_VOLTAGE_ENERGY_STORAGE_PACK_18_HISTORY : UDINT := UDINT#16#FA92; (* < 64146 - HVESP18HIST *)
    PGN_HIGH_VOLTAGE_ENERGY_STORAGE_PACK_18_CONFIGURATION : UDINT := UDINT#16#FA93; (* < 64147 - HVESP18CFG *)
    PGN_HIGH_VOLTAGE_ENERGY_STORAGE_PACK_19_HISTORY : UDINT := UDINT#16#FA94; (* < 64148 - HVESP19HIST *)
    PGN_HIGH_VOLTAGE_ENERGY_STORAGE_PACK_19_CONFIGURATION : UDINT := UDINT#16#FA95; (* < 64149 - HVESP19CFG *)
    PGN_HIGH_VOLTAGE_ENERGY_STORAGE_PACK_20_HISTORY : UDINT := UDINT#16#FA96; (* < 64150 - HVESP20HIST *)
    PGN_HIGH_VOLTAGE_ENERGY_STORAGE_PACK_20_CONFIGURATION : UDINT := UDINT#16#FA97; (* < 64151 - HVESP20CFG *)
    PGN_HIGH_VOLTAGE_ENERGY_STORAGE_PACK_21_HISTORY : UDINT := UDINT#16#FA98; (* < 64152 - HVESP21HIST *)
    PGN_HIGH_VOLTAGE_ENERGY_STORAGE_PACK_21_CONFIGURATION : UDINT := UDINT#16#FA99; (* < 64153 - HVESP21CFG *)
    PGN_HIGH_VOLTAGE_ENERGY_STORAGE_PACK_22_HISTORY : UDINT := UDINT#16#FA9A; (* < 64154 - HVESP22HIST *)
    PGN_HIGH_VOLTAGE_ENERGY_STORAGE_PACK_22_CONFIGURATION : UDINT := UDINT#16#FA9B; (* < 64155 - HVESP22CFG *)
    PGN_HIGH_VOLTAGE_ENERGY_STORAGE_PACK_23_HISTORY : UDINT := UDINT#16#FA9C; (* < 64156 - HVESP23HIST *)
    PGN_HIGH_VOLTAGE_ENERGY_STORAGE_PACK_23_CONFIGURATION : UDINT := UDINT#16#FA9D; (* < 64157 - HVESP23CFG *)
    PGN_HIGH_VOLTAGE_ENERGY_STORAGE_PACK_24_HISTORY : UDINT := UDINT#16#FA9E; (* < 64158 - HVESP24HIST *)
    PGN_HIGH_VOLTAGE_ENERGY_STORAGE_PACK_24_CONFIGURATION : UDINT := UDINT#16#FA9F; (* < 64159 - HVESP24CFG *)
    PGN_HIGH_VOLTAGE_ENERGY_STORAGE_PACK_25_HISTORY : UDINT := UDINT#16#FAA0; (* < 64160 - HVESP25HIST *)
    PGN_HIGH_VOLTAGE_ENERGY_STORAGE_PACK_25_CONFIGURATION : UDINT := UDINT#16#FAA1; (* < 64161 - HVESP25CFG *)
    PGN_HIGH_VOLTAGE_ENERGY_STORAGE_PACK_26_HISTORY : UDINT := UDINT#16#FAA2; (* < 64162 - HVESP26HIST *)
    PGN_HIGH_VOLTAGE_ENERGY_STORAGE_PACK_26_CONFIGURATION : UDINT := UDINT#16#FAA3; (* < 64163 - HVESP26CFG *)
    PGN_AUTOMATED_DRIVING_SYSTEM_CONTROL_2 : UDINT := UDINT#16#FAA4; (* < 64164 - ADSC2 *)
    PGN_DUAL_FUEL_MODE_3 : UDINT := UDINT#16#FAA5; (* < 64165 - DFM3 *)
    PGN_DUAL_FUEL_MODE_2 : UDINT := UDINT#16#FAA6; (* < 64166 - DFM2 *)
    PGN_DUAL_FUEL_MODE_1 : UDINT := UDINT#16#FAA7; (* < 64167 - DFM1 *)
    PGN_TRANSMISSION_1_HISTORY : UDINT := UDINT#16#FAA8; (* < 64168 - T1HIST *)
    PGN_TRANSMISSION_SHAFT_TWIST_INFORMATION : UDINT := UDINT#16#FAA9; (* < 64169 - TSTI *)
    PGN_ELECTRONIC_AUXILIARY_TRANSMISSION_CONTROLLER_2 : UDINT := UDINT#16#FAAA; (* < 64170 - EATC2 *)
    PGN_HIGH_VOLTAGE_ENERGY_STORAGE_PACK_10_CONFIGURATION : UDINT := UDINT#16#FAAB; (* < 64171 - HVESP10CFG *)
    PGN_HIGH_VOLTAGE_ENERGY_STORAGE_PACK_10_HISTORY : UDINT := UDINT#16#FAAC; (* < 64172 - HVESP10HIST *)
    PGN_HIGH_VOLTAGE_ENERGY_STORAGE_PACK_9_CONFIGURATION : UDINT := UDINT#16#FAAD; (* < 64173 - HVESP9CFG *)
    PGN_HIGH_VOLTAGE_ENERGY_STORAGE_PACK_9_HISTORY : UDINT := UDINT#16#FAAE; (* < 64174 - HVESP9HIST *)
    PGN_HIGH_VOLTAGE_ENERGY_STORAGE_PACK_8_CONFIGURATION : UDINT := UDINT#16#FAAF; (* < 64175 - HVESP8CFG *)
    PGN_HIGH_VOLTAGE_ENERGY_STORAGE_PACK_8_HISTORY : UDINT := UDINT#16#FAB0; (* < 64176 - HVESP8HIST *)
    PGN_HIGH_VOLTAGE_ENERGY_STORAGE_PACK_7_CONFIGURATION : UDINT := UDINT#16#FAB1; (* < 64177 - HVESP7CFG *)
    PGN_HIGH_VOLTAGE_ENERGY_STORAGE_PACK_7_HISTORY : UDINT := UDINT#16#FAB2; (* < 64178 - HVESP7HIST *)
    PGN_AUTOSAR_TIME_SYNCHRONIZATION : UDINT := UDINT#16#FAB3; (* < 64179 - CanTSyn *)
    PGN_EV_DC_CHARGING_LIMITS_1 : UDINT := UDINT#16#FAB4; (* < 64180 - EVDCLIM1 *)
    PGN_EVSE_DC_CHARGING_LIMITS_1 : UDINT := UDINT#16#FAB5; (* < 64181 - EVSEDCLIM1 *)
    PGN_EVSE_DC_CHARGING_LIMITS_2 : UDINT := UDINT#16#FAB6; (* < 64182 - EVSEDCLIM2 *)
    PGN_EV_DC_CHARGING_TARGET : UDINT := UDINT#16#FAB7; (* < 64183 - EVDCTGT *)
    PGN_EVSE_DC_STATUS_1 : UDINT := UDINT#16#FAB8; (* < 64184 - EVSEDCS1 *)
    PGN_EVSE_1_CONTACTOR_CMD_1 : UDINT := UDINT#16#FAB9; (* < 64185 - EVSE1CC1 *)
    PGN_EVSE_1_CONTACTOR_STATUS_1 : UDINT := UDINT#16#FABA; (* < 64186 - EVSE1CS1 *)
    PGN_DIRECT_LAMP_CONTROL_COMMAND_3 : UDINT := UDINT#16#FABB; (* < 64187 - DLCC3 *)
    PGN_DIRECT_LAMP_CONTROL_DATA_3 : UDINT := UDINT#16#FABC; (* < 64188 - DLCD3 *)
    PGN_MOTOR_GENERATOR_1_LIFETIME_DATA : UDINT := UDINT#16#FABD; (* < 64189 - MG1LD *)
    PGN_MOTOR_GENERATOR_2_LIFETIME_DATA : UDINT := UDINT#16#FABE; (* < 64190 - MG2LD *)
    PGN_MOTOR_GENERATOR_3_LIFETIME_DATA : UDINT := UDINT#16#FABF; (* < 64191 - MG3LD *)
    PGN_MOTOR_GENERATOR_4_LIFETIME_DATA : UDINT := UDINT#16#FAC0; (* < 64192 - MG4LD *)
    PGN_MOTOR_GENERATOR_5_LIFETIME_DATA : UDINT := UDINT#16#FAC1; (* < 64193 - MG5LD *)
    PGN_MOTOR_GENERATOR_6_LIFETIME_DATA : UDINT := UDINT#16#FAC2; (* < 64194 - MG6LD *)
    PGN_AIR_SUPPLY_PRESSURE_3 : UDINT := UDINT#16#FAC3; (* < 64195 - AIR3 *)
    PGN_EVSE_AC_SUPPLY_VOLTAGE : UDINT := UDINT#16#FAC4; (* < 64196 - EVSEACSV *)
    PGN_EVSE_AC_3_PHASE_LOAD : UDINT := UDINT#16#FAC5; (* < 64197 - EVSEAC3PL *)
    PGN_ELECTRONIC_RETARDER_CONTROLLER_3 : UDINT := UDINT#16#FAC6; (* < 64198 - ERC3 *)
    PGN_ELECTRONIC_TRANSMISSION_CONTROLLER_14 : UDINT := UDINT#16#FAC8; (* < 64200 - ETC14 *)
    PGN_COLLISION_AVOIDANCE_SYSTEM_4 : UDINT := UDINT#16#FACB; (* < 64203 - CXD4 *)
    PGN_COLLISION_AVOIDANCE_SYSTEM_3 : UDINT := UDINT#16#FACC; (* < 64204 - CXD3 *)
    PGN_AFTERTREATMENT_1_SCR_EXHAUST_GAS_PRESSURES_2 : UDINT := UDINT#16#FACD; (* < 64205 - A1SCREGP2 *)
    PGN_PTO_INFORMATION_2 : UDINT := UDINT#16#FACE; (* < 64206 - PTO2 *)
    PGN_EVCC_DIAGNOSTIC_DATA_1 : UDINT := UDINT#16#FACF; (* < 64207 - EVCCD1 *)
    PGN_CAB_DOOR_CONTROL_2 : UDINT := UDINT#16#FAD0; (* < 64208 - CDC2 *)
    PGN_ENGINE_AVERAGE_INFORMATION_2 : UDINT := UDINT#16#FAD1; (* < 64209 - EAI2 *)
    PGN_TURBOCHARGER_INFORMATION_9 : UDINT := UDINT#16#FAD2; (* < 64210 - TCI9 *)
    PGN_AUTOMATED_DRIVING_SYSTEM_CONTROL_1 : UDINT := UDINT#16#FAD3; (* < 64211 - ADSC1 *)
    PGN_EVSE_AC_STATUS_2 : UDINT := UDINT#16#FAD4; (* < 64212 - EVSEACS2 *)
    PGN_EVSE_AC_STATUS_1 : UDINT := UDINT#16#FAD5; (* < 64213 - EVSEACS1 *)
    PGN_EVSE_STATUS_1 : UDINT := UDINT#16#FAD6; (* < 64214 - EVSES1 *)
    PGN_OBJECT_DETECTION_MESSAGE_1_1 : UDINT := UDINT#16#FAD7; (* < 64215 - ODM11 *)
    PGN_OBJECT_DETECTION_MESSAGE_2_1 : UDINT := UDINT#16#FAD8; (* < 64216 - ODM21 *)
    PGN_OBJECT_DETECTION_MESSAGE_2_2 : UDINT := UDINT#16#FAD9; (* < 64217 - ODM22 *)
    PGN_OBJECT_DETECTION_MESSAGE_2_3 : UDINT := UDINT#16#FADA; (* < 64218 - ODM23 *)
    PGN_OBJECT_DETECTION_MESSAGE_2_4 : UDINT := UDINT#16#FADB; (* < 64219 - ODM24 *)
    PGN_OBJECT_DETECTION_MESSAGE_2_5 : UDINT := UDINT#16#FADC; (* < 64220 - ODM25 *)
    PGN_OBJECT_DETECTION_MESSAGE_2_6 : UDINT := UDINT#16#FADD; (* < 64221 - ODM26 *)
    PGN_OBJECT_DETECTION_MESSAGE_2_7 : UDINT := UDINT#16#FADE; (* < 64222 - ODM27 *)
    PGN_OBJECT_DETECTION_MESSAGE_2_8 : UDINT := UDINT#16#FADF; (* < 64223 - ODM28 *)
    PGN_OBJECT_DETECTION_MESSAGE_2_9 : UDINT := UDINT#16#FAE0; (* < 64224 - ODM29 *)
    PGN_OBJECT_DETECTION_MESSAGE_2_10 : UDINT := UDINT#16#FAE1; (* < 64225 - ODM210 *)
    PGN_OBJECT_DETECTION_MESSAGE_2_11 : UDINT := UDINT#16#FAE2; (* < 64226 - ODM211 *)
    PGN_OBJECT_DETECTION_MESSAGE_2_12 : UDINT := UDINT#16#FAE3; (* < 64227 - ODM212 *)
    PGN_OBJECT_DETECTION_MESSAGE_2_13 : UDINT := UDINT#16#FAE4; (* < 64228 - ODM213 *)
    PGN_OBJECT_DETECTION_MESSAGE_2_14 : UDINT := UDINT#16#FAE5; (* < 64229 - ODM214 *)
    PGN_OBJECT_DETECTION_MESSAGE_2_15 : UDINT := UDINT#16#FAE6; (* < 64230 - ODM215 *)
    PGN_OBJECT_DETECTION_MESSAGE_2_16 : UDINT := UDINT#16#FAE7; (* < 64231 - ODM216 *)
    PGN_OBJECT_DETECTION_MESSAGE_2_17 : UDINT := UDINT#16#FAE8; (* < 64232 - ODM217 *)
    PGN_OBJECT_DETECTION_MESSAGE_2_18 : UDINT := UDINT#16#FAE9; (* < 64233 - ODM218 *)
    PGN_OBJECT_DETECTION_MESSAGE_2_19 : UDINT := UDINT#16#FAEA; (* < 64234 - ODM219 *)
    PGN_OBJECT_DETECTION_MESSAGE_2_20 : UDINT := UDINT#16#FAEB; (* < 64235 - ODM220 *)
    PGN_OBJECT_DETECTION_MESSAGE_2_21 : UDINT := UDINT#16#FAEC; (* < 64236 - ODM221 *)
    PGN_TEMPERATURE_SENSING_MODULE_1 : UDINT := UDINT#16#FAED; (* < 64237 - TSM1 *)
    PGN_TEMPERATURE_SENSING_MODULE_2 : UDINT := UDINT#16#FAEE; (* < 64238 - TSM2 *)
    PGN_AFTERTREATMENT_2_SCR_SERVICE_INFORMATION_3 : UDINT := UDINT#16#FAEF; (* < 64239 - A2SCRSI3 *)
    PGN_AFTERTREATMENT_1_SCR_SERVICE_INFORMATION_3 : UDINT := UDINT#16#FAF0; (* < 64240 - A1SCRSI3 *)
    PGN_PSA_TIMES_LIFETIME_HOURS : UDINT := UDINT#16#FAF1; (* < 64241 - PSATL *)
    PGN_PSA_TIMES_STORED_100_HOURS : UDINT := UDINT#16#FAF2; (* < 64242 - PSATS *)
    PGN_PSA_TIMES_ACTIVE_100_HOURS : UDINT := UDINT#16#FAF3; (* < 64243 - PSATA *)
    PGN_HYBRID_CHARGE_DEPLETING_OR_INCREASING_OPERATION_LIFETIME_HOURS : UDINT := UDINT#16#FAF4; (* < 64244 - HCDIOL *)
    PGN_HYBRID_CHARGE_DEPLETING_OR_INCREASING_OPERATION_STORED_100_HOURS : UDINT := UDINT#16#FAF5; (* < 64245 - HCDIOS *)
    PGN_HYBRID_CHARGE_DEPLETING_OR_INCREASING_OPERATION_ACTIVE_100_HOURS : UDINT := UDINT#16#FAF6; (* < 64246 - HCDIOA *)
    PGN_AFTERTREATMENT_1_HISTORICAL_INFORMATION_3 : UDINT := UDINT#16#FAF7; (* < 64247 - AT1HI3 *)
    PGN_ENGINE_MAXIMUM_NET_TORQUE_MAP : UDINT := UDINT#16#FAF8; (* < 64248 - ENGMXT *)
    PGN_AFTERTREATMENT_1_SCR_2_NOX_MASS_AND_NH3_STORAGE : UDINT := UDINT#16#FAF9; (* < 64249 - ATNXMS2 *)
    PGN_AFTERTREATMENT_1_SCR_1_NOX_MASS_AND_NH3_STORAGE : UDINT := UDINT#16#FAFA; (* < 64250 - ATNXMS1 *)
    PGN_EVAPORATIVE_SYSTEM_PRESSURE_AND_CONTROL : UDINT := UDINT#16#FAFB; (* < 64251 - ESPC *)
    PGN_GHG_TRACKING_LIFETIME_ARRAY_DATA : UDINT := UDINT#16#FAFC; (* < 64252 - GHGTL *)
    PGN_GHG_TRACKING_STORED_100_HOUR_ARRAY_DATA : UDINT := UDINT#16#FAFD; (* < 64253 - GHGTS *)
    PGN_GHG_TRACKING_ACTIVE_100_HOUR_ARRAY_DATA : UDINT := UDINT#16#FAFE; (* < 64254 - GHGTA *)
    PGN_GREEN_HOUSE_GAS_STORED_100_HOUR_ACTIVE_TECHNOLOGY_TRACKING : UDINT := UDINT#16#FAFF; (* < 64255 - GHGTTS *)
    PGN_GREEN_HOUSE_GAS_ACTIVE_100_HOUR_ACTIVE_TECHNOLOGY_TRACKING : UDINT := UDINT#16#FB00; (* < 64256 - GHGTTA *)
    PGN_GREEN_HOUSE_GAS_LIFETIME_ACTIVE_TECHNOLOGY_TRACKING : UDINT := UDINT#16#FB01; (* < 64257 - GHGTTL *)
    PGN_NOX_TRACKING_ENGINE_ACTIVITY_LIFETIME_FUEL_CONSUMPTION_BINS : UDINT := UDINT#16#FB02; (* < 64258 - NTFCEA *)
    PGN_NOX_TRACKING_ENGINE_ACTIVITY_LIFETIME_ENGINE_RUN_TIME_BINS : UDINT := UDINT#16#FB03; (* < 64259 - NTEHEA *)
    PGN_NOX_TRACKING_ENGINE_ACTIVITY_LIFETIME_VEHICLE_DISTANCE_BINS : UDINT := UDINT#16#FB04; (* < 64260 - NTVMEA *)
    PGN_NOX_TRACKING_ENGINE_ACTIVITY_LIFETIME_ENGINE_OUTPUT_ENERGY_BINS : UDINT := UDINT#16#FB05; (* < 64261 - NTEEEA *)
    PGN_NOX_TRACKING_VALID_NOX_LIFETIME_FUEL_CONSUMPTION_BINS : UDINT := UDINT#16#FB06; (* < 64262 - NTFCV *)
    PGN_NOX_TRACKING_VALID_NOX_LIFETIME_ENGINE_RUN_TIME_BINS : UDINT := UDINT#16#FB07; (* < 64263 - NTEHV *)
    PGN_NOX_TRACKING_VALID_NOX_LIFETIME_VEHICLE_DISTANCE_BINS : UDINT := UDINT#16#FB08; (* < 64264 - NTVMV *)
    PGN_NOX_TRACKING_VALID_NOX_LIFETIME_ENGINE_OUTPUT_ENERGY_BINS : UDINT := UDINT#16#FB09; (* < 64265 - NTEEV *)
    PGN_NOX_TRACKING_VALID_NOX_LIFETIME_ENGINE_OUT_NOX_MASS_BINS : UDINT := UDINT#16#FB0A; (* < 64266 - NTENV *)
    PGN_NOX_TRACKING_VALID_NOX_LIFETIME_SYSTEM_OUT_NOX_MASS_BINS : UDINT := UDINT#16#FB0B; (* < 64267 - NTSNV *)
    PGN_NOX_TRACKING_STORED_100_HOUR_FUEL_CONSUMPTION_BINS : UDINT := UDINT#16#FB0C; (* < 64268 - NTFCS *)
    PGN_NOX_TRACKING_STORED_100_HOUR_ENGINE_RUN_TIME_BINS : UDINT := UDINT#16#FB0D; (* < 64269 - NTEHS *)
    PGN_NOX_TRACKING_STORED_100_HOUR_VEHICLE_DISTANCE_BINS : UDINT := UDINT#16#FB0E; (* < 64270 - NTVMS *)
    PGN_NOX_TRACKING_STORED_100_HOUR_ENGINE_OUTPUT_ENERGY_BINS : UDINT := UDINT#16#FB0F; (* < 64271 - NTEES *)
    PGN_NOX_TRACKING_STORED_100_HOUR_ENGINE_OUT_NOX_MASS_BINS : UDINT := UDINT#16#FB10; (* < 64272 - NTENS *)
    PGN_NOX_TRACKING_STORED_100_HOUR_SYSTEM_OUT_NOX_MASS_BINS : UDINT := UDINT#16#FB11; (* < 64273 - NTSNS *)
    PGN_NOX_TRACKING_ACTIVE_100_HOUR_FUEL_CONSUMPTION_BINS : UDINT := UDINT#16#FB12; (* < 64274 - NTFCA *)
    PGN_NOX_TRACKING_ACTIVE_100_HOUR_ENGINE_RUN_TIME_BINS : UDINT := UDINT#16#FB13; (* < 64275 - NTEHA *)
    PGN_NOX_TRACKING_ACTIVE_100_HOUR_VEHICLE_DISTANCE_BINS : UDINT := UDINT#16#FB14; (* < 64276 - NTVMA *)
    PGN_NOX_TRACKING_ACTIVE_100_HOUR_ENGINE_OUTPUT_ENERGY_BINS : UDINT := UDINT#16#FB15; (* < 64277 - NTEEA *)
    PGN_NOX_TRACKING_ACTIVE_100_HOUR_ENGINE_OUT_NOX_MASS_BINS : UDINT := UDINT#16#FB16; (* < 64278 - NTENA *)
    PGN_NOX_TRACKING_ACTIVE_100_HOUR_SYSTEM_OUT_NOX_MASS_BINS : UDINT := UDINT#16#FB17; (* < 64279 - NTSNA *)
    PGN_MOTOR_GENERATOR_6_INVERTER_CONTROL_2 : UDINT := UDINT#16#FB18; (* < 64280 - MG6IC2 *)
    PGN_MOTOR_GENERATOR_6_INVERTER_LIMITS_REQUEST_POWER : UDINT := UDINT#16#FB19; (* < 64281 - MG6IRP *)
    PGN_MOTOR_GENERATOR_6_INVERTER_LIMITS_REQUEST_MECHANICAL : UDINT := UDINT#16#FB1A; (* < 64282 - MG6ILRM *)
    PGN_MOTOR_GENERATOR_6_INVERTER_LIMITS_REQUEST_DC_SIDE : UDINT := UDINT#16#FB1B; (* < 64283 - MG6ILRDC *)
    PGN_MOTOR_GENERATOR_6_INVERTER_ISOLATION_INTEGRITY_REQUEST : UDINT := UDINT#16#FB1C; (* < 64284 - MG6IIR *)
    PGN_MOTOR_GENERATOR_5_INVERTER_CONTROL_2 : UDINT := UDINT#16#FB1D; (* < 64285 - MG5IC2 *)
    PGN_MOTOR_GENERATOR_5_INVERTER_LIMITS_REQUEST_POWER : UDINT := UDINT#16#FB1E; (* < 64286 - MG5IRP *)
    PGN_MOTOR_GENERATOR_5_INVERTER_LIMITS_REQUEST_MECHANICAL : UDINT := UDINT#16#FB1F; (* < 64287 - MG5ILRM *)
    PGN_MOTOR_GENERATOR_5_INVERTER_LIMITS_REQUEST_DC_SIDE : UDINT := UDINT#16#FB20; (* < 64288 - MG5ILRDC *)
    PGN_MOTOR_GENERATOR_5_INVERTER_ISOLATION_INTEGRITY_REQUEST : UDINT := UDINT#16#FB21; (* < 64289 - MG5IIR *)
    PGN_MOTOR_GENERATOR_4_INVERTER_CONTROL_2 : UDINT := UDINT#16#FB22; (* < 64290 - MG4IC2 *)
    PGN_MOTOR_GENERATOR_4_INVERTER_LIMITS_REQUEST_POWER : UDINT := UDINT#16#FB23; (* < 64291 - MG4IRP *)
    PGN_MOTOR_GENERATOR_4_INVERTER_LIMITS_REQUEST_MECHANICAL : UDINT := UDINT#16#FB24; (* < 64292 - MG4ILRM *)
    PGN_MOTOR_GENERATOR_4_INVERTER_LIMITS_REQUEST_DC_SIDE : UDINT := UDINT#16#FB25; (* < 64293 - MG4ILRDC *)
    PGN_MOTOR_GENERATOR_4_INVERTER_ISOLATION_INTEGRITY_REQUEST : UDINT := UDINT#16#FB26; (* < 64294 - MG4IIR *)
    PGN_MOTOR_GENERATOR_3_INVERTER_CONTROL_2 : UDINT := UDINT#16#FB27; (* < 64295 - MG3IC2 *)
    PGN_MOTOR_GENERATOR_3_INVERTER_LIMITS_REQUEST_POWER : UDINT := UDINT#16#FB28; (* < 64296 - MG3IRP *)
    PGN_MOTOR_GENERATOR_3_INVERTER_LIMITS_REQUEST_MECHANICAL : UDINT := UDINT#16#FB29; (* < 64297 - MG3ILRM *)
    PGN_MOTOR_GENERATOR_3_INVERTER_LIMITS_REQUEST_DC_SIDE : UDINT := UDINT#16#FB2A; (* < 64298 - MG3ILRDC *)
    PGN_MOTOR_GENERATOR_3_INVERTER_ISOLATION_INTEGRITY_REQUEST : UDINT := UDINT#16#FB2B; (* < 64299 - MG3IIR *)
    PGN_DIAGNOSTIC_READINESS_4 : UDINT := UDINT#16#FB2C; (* < 64300 - DM59 *)
    PGN_TURBOCHARGER_INFORMATION_8 : UDINT := UDINT#16#FB2D; (* < 64301 - TCI8 *)
    PGN_WINCH_INFORMATION_2 : UDINT := UDINT#16#FB2E; (* < 64302 - WINCH2 *)
    PGN_MOTOR_GENERATOR_6_INVERTER_REFERENCE_1 : UDINT := UDINT#16#FB2F; (* < 64303 - MG6IR1 *)
    PGN_MOTOR_GENERATOR_6_INVERTER_STATUS_1 : UDINT := UDINT#16#FB30; (* < 64304 - MG6IS1 *)
    PGN_MOTOR_GENERATOR_6_INVERTER_REFERENCE_2 : UDINT := UDINT#16#FB31; (* < 64305 - MG6IR2 *)
    PGN_MOTOR_GENERATOR_6_INVERTER_TEMPERATURE : UDINT := UDINT#16#FB32; (* < 64306 - MG6IT *)
    PGN_MOTOR_GENERATOR_6_INVERTER_MOTOR_TEMPERATURE : UDINT := UDINT#16#FB33; (* < 64307 - MG6IMT *)
    PGN_MOTOR_GENERATOR_6_INVERTER_ISOLATION_INTEGRITY : UDINT := UDINT#16#FB34; (* < 64308 - MG6II *)
    PGN_MOTOR_GENERATOR_6_INVERTER_ACTIVE_POWER_LIMITS : UDINT := UDINT#16#FB35; (* < 64309 - MG6IAPL *)
    PGN_MOTOR_GENERATOR_5_INVERTER_REFERENCE_1 : UDINT := UDINT#16#FB36; (* < 64310 - MG5IR1 *)
    PGN_MOTOR_GENERATOR_5_INVERTER_STATUS_1 : UDINT := UDINT#16#FB37; (* < 64311 - MG5IS1 *)
    PGN_MOTOR_GENERATOR_5_INVERTER_REFERENCE_2 : UDINT := UDINT#16#FB38; (* < 64312 - MG5IR2 *)
    PGN_MOTOR_GENERATOR_5_INVERTER_TEMPERATURE : UDINT := UDINT#16#FB39; (* < 64313 - MG5IT *)
    PGN_MOTOR_GENERATOR_5_INVERTER_MOTOR_TEMPERATURE : UDINT := UDINT#16#FB3A; (* < 64314 - MG5IMT *)
    PGN_MOTOR_GENERATOR_5_INVERTER_ISOLATION_INTEGRITY : UDINT := UDINT#16#FB3B; (* < 64315 - MG5II *)
    PGN_MOTOR_GENERATOR_5_INVERTER_ACTIVE_POWER_LIMITS : UDINT := UDINT#16#FB3C; (* < 64316 - MG5IAPL *)
    PGN_MOTOR_GENERATOR_4_INVERTER_REFERENCE_1 : UDINT := UDINT#16#FB3D; (* < 64317 - MG4IR1 *)
    PGN_MOTOR_GENERATOR_4_INVERTER_STATUS_1 : UDINT := UDINT#16#FB3E; (* < 64318 - MG4IS1 *)
    PGN_MOTOR_GENERATOR_4_INVERTER_REFERENCE_2 : UDINT := UDINT#16#FB3F; (* < 64319 - MG4IR2 *)
    PGN_MOTOR_GENERATOR_4_INVERTER_TEMPERATURE : UDINT := UDINT#16#FB40; (* < 64320 - MG4IT *)
    PGN_MOTOR_GENERATOR_4_INVERTER_MOTOR_TEMPERATURE : UDINT := UDINT#16#FB41; (* < 64321 - MG4IMT *)
    PGN_MOTOR_GENERATOR_4_INVERTER_ISOLATION_INTEGRITY : UDINT := UDINT#16#FB42; (* < 64322 - MG4II *)
    PGN_MOTOR_GENERATOR_4_INVERTER_ACTIVE_POWER_LIMITS : UDINT := UDINT#16#FB43; (* < 64323 - MG4IAPL *)
    PGN_MOTOR_GENERATOR_3_INVERTER_REFERENCE_1 : UDINT := UDINT#16#FB44; (* < 64324 - MG3IR1 *)
    PGN_MOTOR_GENERATOR_3_INVERTER_STATUS_1 : UDINT := UDINT#16#FB45; (* < 64325 - MG3IS1 *)
    PGN_MOTOR_GENERATOR_3_INVERTER_REFERENCE_2 : UDINT := UDINT#16#FB46; (* < 64326 - MG3IR2 *)
    PGN_MOTOR_GENERATOR_3_INVERTER_TEMPERATURE : UDINT := UDINT#16#FB47; (* < 64327 - MG3IT *)
    PGN_MOTOR_GENERATOR_3_INVERTER_MOTOR_TEMPERATURE : UDINT := UDINT#16#FB48; (* < 64328 - MG3IMT *)
    PGN_MOTOR_GENERATOR_3_INVERTER_ISOLATION_INTEGRITY : UDINT := UDINT#16#FB49; (* < 64329 - MG3II *)
    PGN_MOTOR_GENERATOR_3_INVERTER_ACTIVE_POWER_LIMITS : UDINT := UDINT#16#FB4A; (* < 64330 - MG3IAPL *)
    PGN_AUTOMATED_DRIVING_SYSTEM_STATUS_1 : UDINT := UDINT#16#FB4B; (* < 64331 - ADSS1 *)
    PGN_CAB_CLIMATE_SYSTEM_INFORMATION_2 : UDINT := UDINT#16#FB4C; (* < 64332 - CCSI2 *)
    PGN_MAINTENANCE_INFORMATION_1 : UDINT := UDINT#16#FB4D; (* < 64333 - MI1 *)
    PGN_HOIST_CONTROL_INFORMATION : UDINT := UDINT#16#FB4E; (* < 64334 - HCI1 *)
    PGN_HIGH_VOLTAGE_ENERGY_STORAGE_PACK_6_HISTORY : UDINT := UDINT#16#FB4F; (* < 64335 - HVESP6HIST *)
    PGN_HIGH_VOLTAGE_ENERGY_STORAGE_PACK_6_CONFIGURATION : UDINT := UDINT#16#FB50; (* < 64336 - HVESP6CFG *)
    PGN_HIGH_VOLTAGE_ENERGY_STORAGE_PACK_5_HISTORY : UDINT := UDINT#16#FB51; (* < 64337 - HVESP5HIST *)
    PGN_HIGH_VOLTAGE_ENERGY_STORAGE_PACK_5_CONFIGURATION : UDINT := UDINT#16#FB52; (* < 64338 - HVESP5CFG *)
    PGN_HIGH_VOLTAGE_ENERGY_STORAGE_PACK_4_HISTORY : UDINT := UDINT#16#FB53; (* < 64339 - HVESP4HIST *)
    PGN_HIGH_VOLTAGE_ENERGY_STORAGE_PACK_4_CONFIGURATION : UDINT := UDINT#16#FB54; (* < 64340 - HVESP4CFG *)
    PGN_HIGH_VOLTAGE_ENERGY_STORAGE_PACK_3_HISTORY : UDINT := UDINT#16#FB55; (* < 64341 - HVESP3HIST *)
    PGN_HIGH_VOLTAGE_ENERGY_STORAGE_PACK_3_CONFIGURATION : UDINT := UDINT#16#FB56; (* < 64342 - HVESP3CFG *)
    PGN_HIGH_VOLTAGE_ENERGY_STORAGE_PACK_2_HISTORY : UDINT := UDINT#16#FB57; (* < 64343 - HVESP2HIST *)
    PGN_HIGH_VOLTAGE_ENERGY_STORAGE_PACK_2_CONFIGURATION : UDINT := UDINT#16#FB58; (* < 64344 - HVESP2CFG *)
    PGN_HIGH_VOLTAGE_ENERGY_STORAGE_PACK_1_HISTORY : UDINT := UDINT#16#FB59; (* < 64345 - HVESP1HIST *)
    PGN_HIGH_VOLTAGE_ENERGY_STORAGE_PACK_1_CONFIGURATION : UDINT := UDINT#16#FB5A; (* < 64346 - HVESP1CFG *)
    PGN_VEHICLE_FIRE_SUPPRESSION_SYSTEM_MODULE_1_DETECTOR_DATA : UDINT := UDINT#16#FB5B; (* < 64347 - VFSSM1DET *)
    PGN_VEHICLE_FIRE_SUPPRESSION_SYSTEM_MODULE_2_DETECTOR_DATA : UDINT := UDINT#16#FB5C; (* < 64348 - VFSSM2DET *)
    PGN_VEHICLE_FIRE_SUPPRESSION_SYSTEM_MODULE_3_DETECTOR_DATA : UDINT := UDINT#16#FB5D; (* < 64349 - VFSSM3DET *)
    PGN_VEHICLE_FIRE_SUPPRESSION_SYSTEM_MODULE_4_DETECTOR_DATA : UDINT := UDINT#16#FB5E; (* < 64350 - VFSSM4DET *)
    PGN_VEHICLE_FIRE_SUPPRESSION_SYSTEM_MODULE_1_AUXILIARY_DATA : UDINT := UDINT#16#FB5F; (* < 64351 - VFSSM1AUX *)
    PGN_VEHICLE_FIRE_SUPPRESSION_SYSTEM_MODULE_2_AUXILIARY_DATA : UDINT := UDINT#16#FB60; (* < 64352 - VFSSM2AUX *)
    PGN_VEHICLE_FIRE_SUPPRESSION_SYSTEM_MODULE_3_AUXILIARY_DATA : UDINT := UDINT#16#FB61; (* < 64353 - VFSSM3AUX *)
    PGN_VEHICLE_FIRE_SUPPRESSION_SYSTEM_MODULE_4_AUXILIARY_DATA : UDINT := UDINT#16#FB62; (* < 64354 - VFSSM4AUX *)
    PGN_VEHICLE_FIRE_SUPPRESSION_SYSTEM_MODULE_1_NAMES : UDINT := UDINT#16#FB63; (* < 64355 - VFSSM1NAMES *)
    PGN_VEHICLE_FIRE_SUPPRESSION_SYSTEM_MODULE_2_NAMES : UDINT := UDINT#16#FB64; (* < 64356 - VFSSM2NAMES *)
    PGN_VEHICLE_FIRE_SUPPRESSION_SYSTEM_MODULE_3_NAMES : UDINT := UDINT#16#FB65; (* < 64357 - VFSSM3NAMES *)
    PGN_VEHICLE_FIRE_SUPPRESSION_SYSTEM_MODULE_4_NAMES : UDINT := UDINT#16#FB66; (* < 64358 - VFSSM4NAMES *)
    PGN_MOTOR_GENERATOR_2_INVERTER_ACTIVE_POWER_LIMITS : UDINT := UDINT#16#FB67; (* < 64359 - MG2IAPL *)
    PGN_MOTOR_GENERATOR_2_INVERTER_ISOLATION_INTEGRITY : UDINT := UDINT#16#FB68; (* < 64360 - MG2II *)
    PGN_MOTOR_GENERATOR_1_INVERTER_ACTIVE_POWER_LIMITS : UDINT := UDINT#16#FB69; (* < 64361 - MG1IAPL *)
    PGN_MOTOR_GENERATOR_1_INVERTER_ISOLATION_INTEGRITY : UDINT := UDINT#16#FB6A; (* < 64362 - MG1II *)
    PGN_HIGH_VOLTAGE_BUS_INFORMATION : UDINT := UDINT#16#FB6B; (* < 64363 - HVBI *)
    PGN_MOTOR_GENERATOR_2_INVERTER_REFERENCE_1 : UDINT := UDINT#16#FB6C; (* < 64364 - MG2IR1 *)
    PGN_MOTOR_GENERATOR_2_INVERTER_STATUS_1 : UDINT := UDINT#16#FB6D; (* < 64365 - MG2IS1 *)
    PGN_MOTOR_GENERATOR_2_INVERTER_REFERENCE_2 : UDINT := UDINT#16#FB6E; (* < 64366 - MG2IR2 *)
    PGN_MOTOR_GENERATOR_2_INVERTER_TEMPERATURE : UDINT := UDINT#16#FB6F; (* < 64367 - MG2IT *)
    PGN_MOTOR_GENERATOR_2_INVERTER_MOTOR_TEMPERATURE : UDINT := UDINT#16#FB70; (* < 64368 - MG2IMT *)
    PGN_MOTOR_GENERATOR_1_INVERTER_MOTOR_TEMPERATURE : UDINT := UDINT#16#FB71; (* < 64369 - MG1IMT *)
    PGN_MOTOR_GENERATOR_1_INVERTER_TEMPERATURE : UDINT := UDINT#16#FB72; (* < 64370 - MG1IT *)
    PGN_MOTOR_GENERATOR_1_INVERTER_REFERENCE_2 : UDINT := UDINT#16#FB73; (* < 64371 - MG1IR2 *)
    PGN_MOTOR_GENERATOR_1_INVERTER_STATUS_1 : UDINT := UDINT#16#FB74; (* < 64372 - MG1IS1 *)
    PGN_MOTOR_GENERATOR_1_INVERTER_REFERENCE_1 : UDINT := UDINT#16#FB75; (* < 64373 - MG1IR1 *)
    PGN_PERSONNEL_DETECT_STATUS : UDINT := UDINT#16#FB76; (* < 64374 - PDS *)
    PGN_ENGINE_CYLINDER_PRESSURE_GAMMA_1 : UDINT := UDINT#16#FB77; (* < 64375 - ECPG1 *)
    PGN_ENGINE_CYLINDER_PRESSURE_GAMMA_2 : UDINT := UDINT#16#FB78; (* < 64376 - ECPG2 *)
    PGN_ENGINE_CYLINDER_PRESSURE_GAMMA_3 : UDINT := UDINT#16#FB79; (* < 64377 - ECPG3 *)
    PGN_ENGINE_CYLINDER_PRESSURE_GAMMA_4 : UDINT := UDINT#16#FB7A; (* < 64378 - ECPG4 *)
    PGN_ENGINE_CYLINDER_PRESSURE_GAMMA_5 : UDINT := UDINT#16#FB7B; (* < 64379 - ECPG5 *)
    PGN_WAKE_UP_AND_SLEEP : UDINT := UDINT#16#FB7C; (* < 64380 - WAKE *)
    PGN_ELECTRIFIED_ACCESSORY_GENERATOR_COOLANT_PUMP_STATUS_1 : UDINT := UDINT#16#FB7D; (* < 64381 - EAGCPS1 *)
    PGN_ELECTRIFIED_ACCESSORY_GENERATOR_COOLANT_FAN_STATUS_1 : UDINT := UDINT#16#FB7E; (* < 64382 - EAGCFS1 *)
    PGN_WELL_STIMULATION_PUMP_SYSTEM_FILTER_INFORMATION : UDINT := UDINT#16#FB7F; (* < 64383 - WSPF *)
    PGN_PTO_GOVERNOR_CONFIGURATION : UDINT := UDINT#16#FB80; (* < 64384 - PTOGC *)
    PGN_ON_BOARD_PROGRAMMING_2 : UDINT := UDINT#16#FB81; (* < 64385 - OBP2 *)
    PGN_PRIMARY_OR_REAR_HITCH_YAW : UDINT := UDINT#16#FB82; (* < 64386 - RHY *)
    PGN_SECONDARY_OR_FRONT_HITCH_YAW : UDINT := UDINT#16#FB83; (* < 64387 - FHY *)
    PGN_OPERATOR_STATUS : UDINT := UDINT#16#FB84; (* < 64388 - OPSTAT *)
    PGN_ENGINE_IDLE_MANAGEMENT_INFORMATION : UDINT := UDINT#16#FB85; (* < 64389 - EIMI *)
    PGN_ALCOHOL_INTERLOCK_TO_VEHICLE : UDINT := UDINT#16#FB86; (* < 64390 - AITOV *)
    PGN_VEHICLE_TO_ALCOHOL_INTERLOCK : UDINT := UDINT#16#FB87; (* < 64391 - VTOAI *)
    PGN_MARINE_CONTROL_INFORMATION_3 : UDINT := UDINT#16#FB88; (* < 64392 - MCI3 *)
    PGN_ENGINE_FLUID_LEVEL_PRESSURE_13 : UDINT := UDINT#16#FB89; (* < 64393 - EFL/P13 *)
    PGN_HIGH_VOLTAGE_ENERGY_STORAGE_SYSTEM_DATA_11 : UDINT := UDINT#16#FB8A; (* < 64394 - HVESSD11 *)
    PGN_ECONOMY_MODE_INACTIVE_HOURS : UDINT := UDINT#16#FB8B; (* < 64395 - EMIH *)
    PGN_ECONOMY_MODE_ESTIMATED_INSTANTANEOUS_FUEL_SAVINGS_RATE : UDINT := UDINT#16#FB8C; (* < 64396 - EMEIFSR *)
    PGN_ECONOMY_MODE_ACTIVE_HOURS : UDINT := UDINT#16#FB8D; (* < 64397 - EMAH *)
    PGN_ECONOMY_MODE_FUEL_USED : UDINT := UDINT#16#FB8E; (* < 64398 - EMFU *)
    PGN_ECONOMY_MODE_ESTIMATED_FUEL_SAVINGS : UDINT := UDINT#16#FB8F; (* < 64399 - EMEFS *)
    PGN_DC_DC_CONVERTER_4_VOLTAGE : UDINT := UDINT#16#FB90; (* < 64400 - DCDC4V *)
    PGN_DC_DC_CONVERTER_3_VOLTAGE : UDINT := UDINT#16#FB91; (* < 64401 - DCDC3V *)
    PGN_DC_DC_CONVERTER_2_VOLTAGE : UDINT := UDINT#16#FB92; (* < 64402 - DCDC2V *)
    PGN_DC_DC_CONVERTER_1_VOLTAGE : UDINT := UDINT#16#FB93; (* < 64403 - DCDC1V *)
    PGN_ELECTRONIC_ENGINE_CONTROLLER_22 : UDINT := UDINT#16#FB94; (* < 64404 - EEC22 *)
    PGN_ENGINE_HOURS_2 : UDINT := UDINT#16#FB95; (* < 64405 - HOURS2 *)
    PGN_ENGINE_INFORMATION_3 : UDINT := UDINT#16#FB96; (* < 64406 - EI3 *)
    PGN_VEHICLE_ELECTRICAL_POWER_15 : UDINT := UDINT#16#FB97; (* < 64407 - VEP15 *)
    PGN_EXHAUST_OXYGEN_2 : UDINT := UDINT#16#FB98; (* < 64408 - EO2 *)
    PGN_DC_AC_ACCESSORY_INVERTER_1_TEMPERATURES : UDINT := UDINT#16#FB99; (* < 64409 - DCAC_AI1_T *)
    PGN_DC_AC_ACCESSORY_INVERTER_1_DC_SIDE_LIMITS : UDINT := UDINT#16#FB9A; (* < 64410 - DCAC_AI1_DCL *)
    PGN_DC_AC_ACCESSORY_INVERTER_1_AC_SIDE_LIMITS : UDINT := UDINT#16#FB9B; (* < 64411 - DCAC_AI1_ACL *)
    PGN_DC_AC_ACCESSORY_INVERTER_1_CONFIGURATION_1 : UDINT := UDINT#16#FB9C; (* < 64412 - DCAC_AI1_CFG1 *)
    PGN_DC_AC_ACCESSORY_INVERTER_1_LIFETIME_DATA : UDINT := UDINT#16#FB9D; (* < 64413 - DCAC_AI1_LD *)
    PGN_DC_AC_ACCESSORY_INVERTER_2_TEMPERATURES : UDINT := UDINT#16#FB9E; (* < 64414 - DCAC_AI2_T *)
    PGN_DC_AC_ACCESSORY_INVERTER_2_DC_SIDE_LIMITS : UDINT := UDINT#16#FB9F; (* < 64415 - DCAC_AI2_DCL *)
    PGN_DC_AC_ACCESSORY_INVERTER_2_AC_SIDE_LIMITS : UDINT := UDINT#16#FBA0; (* < 64416 - DCAC_AI2_ACL *)
    PGN_DC_AC_ACCESSORY_INVERTER_2_CONFIGURATION_1 : UDINT := UDINT#16#FBA1; (* < 64417 - DCAC_AI2_CFG1 *)
    PGN_DC_AC_ACCESSORY_INVERTER_2_LIFETIME_DATA : UDINT := UDINT#16#FBA2; (* < 64418 - DCAC_AI2_LD *)
    PGN_DC_AC_ACCESSORY_INVERTER_3_TEMPERATURES : UDINT := UDINT#16#FBA3; (* < 64419 - DCAC_AI3_T *)
    PGN_DC_AC_ACCESSORY_INVERTER_3_DC_SIDE_LIMITS : UDINT := UDINT#16#FBA4; (* < 64420 - DCAC_AI3_DCL *)
    PGN_DC_AC_ACCESSORY_INVERTER_3_AC_SIDE_LIMITS : UDINT := UDINT#16#FBA5; (* < 64421 - DCAC_AI3_ACL *)
    PGN_DC_AC_ACCESSORY_INVERTER_3_CONFIGURATION_1 : UDINT := UDINT#16#FBA6; (* < 64422 - DCAC_AI3_CFG1 *)
    PGN_DC_AC_ACCESSORY_INVERTER_3_LIFETIME_DATA : UDINT := UDINT#16#FBA7; (* < 64423 - DCAC_AI3_LD *)
    PGN_DC_AC_ACCESSORY_INVERTER_4_TEMPERATURES : UDINT := UDINT#16#FBA8; (* < 64424 - DCAC_AI4_T *)
    PGN_DC_AC_ACCESSORY_INVERTER_4_DC_SIDE_LIMITS : UDINT := UDINT#16#FBA9; (* < 64425 - DCAC_AI4_DCL *)
    PGN_DC_AC_ACCESSORY_INVERTER_4_AC_SIDE_LIMITS : UDINT := UDINT#16#FBAA; (* < 64426 - DCAC_AI4_ACL *)
    PGN_DC_AC_ACCESSORY_INVERTER_4_CONFIGURATION_1 : UDINT := UDINT#16#FBAB; (* < 64427 - DCAC_AI4_CFG1 *)
    PGN_DC_AC_ACCESSORY_INVERTER_4_LIFETIME_DATA : UDINT := UDINT#16#FBAC; (* < 64428 - DCAC_AI4_LD *)
    PGN_DC_AC_ACCESSORY_INVERTER_5_TEMPERATURES : UDINT := UDINT#16#FBAD; (* < 64429 - DCAC_AI5_T *)
    PGN_DC_AC_ACCESSORY_INVERTER_5_DC_SIDE_LIMITS : UDINT := UDINT#16#FBAE; (* < 64430 - DCAC_AI5_DCL *)
    PGN_DC_AC_ACCESSORY_INVERTER_5_AC_SIDE_LIMITS : UDINT := UDINT#16#FBAF; (* < 64431 - DCAC_AI5_ACL *)
    PGN_DC_AC_ACCESSORY_INVERTER_5_CONFIGURATION_1 : UDINT := UDINT#16#FBB0; (* < 64432 - DCAC_AI5_CFG1 *)
    PGN_DC_AC_ACCESSORY_INVERTER_5_LIFETIME_DATA : UDINT := UDINT#16#FBB1; (* < 64433 - DCAC_AI5_LD *)
    PGN_WELL_STIMULATION_PUMP_SENSOR_CALIBRATION_STATUS : UDINT := UDINT#16#FBB2; (* < 64434 - WSPSCS *)
    PGN_WELL_STIMULATION_PUMP_FLUID_VOLUME : UDINT := UDINT#16#FBB3; (* < 64435 - WSPFV *)
    PGN_WELL_STIMULATION_PUMP_SERIAL_NUMBER : UDINT := UDINT#16#FBB4; (* < 64436 - WSPSN *)
    PGN_WELL_STIMULATION_PUMP_TRIP_HOURS : UDINT := UDINT#16#FBB5; (* < 64437 - WSPH2 *)
    PGN_AFTERTREATMENT_1_OUTLET_GAS_4 : UDINT := UDINT#16#FBB6; (* < 64438 - AT1OG4 *)
    PGN_AFTERTREATMENT_1_INTAKE_GAS_4 : UDINT := UDINT#16#FBB7; (* < 64439 - AT1IG4 *)
    PGN_DC_DC_CONVERTER_4_LIFETIME_DATA : UDINT := UDINT#16#FBB8; (* < 64440 - DCDC4LD *)
    PGN_DC_DC_CONVERTER_4_CONFIGURATION_1 : UDINT := UDINT#16#FBB9; (* < 64441 - DCDC4CFG1 *)
    PGN_DC_DC_CONVERTER_4_SLI_BATTERY_LIMITS : UDINT := UDINT#16#FBBA; (* < 64442 - DCDC4SBL *)
    PGN_DC_DC_CONVERTER_4_TEMPERATURES : UDINT := UDINT#16#FBBB; (* < 64443 - DCDC4T *)
    PGN_DC_DC_CONVERTER_4_LOW_SIDE_LIMITS : UDINT := UDINT#16#FBBC; (* < 64444 - DCDC4LL *)
    PGN_DC_DC_CONVERTER_4_HIGH_SIDE_LIMITS : UDINT := UDINT#16#FBBD; (* < 64445 - DCDC4HL *)
    PGN_DC_DC_CONVERTER_3_LIFETIME_DATA : UDINT := UDINT#16#FBBE; (* < 64446 - DCDC3LD *)
    PGN_DC_DC_CONVERTER_3_CONFIGURATION_1 : UDINT := UDINT#16#FBBF; (* < 64447 - DCDC3CFG1 *)
    PGN_DC_DC_CONVERTER_3_SLI_BATTERY_LIMITS : UDINT := UDINT#16#FBC0; (* < 64448 - DCDC3SBL *)
    PGN_DC_DC_CONVERTER_3_TEMPERATURES : UDINT := UDINT#16#FBC1; (* < 64449 - DCDC3T *)
    PGN_DC_DC_CONVERTER_3_LOW_SIDE_LIMITS : UDINT := UDINT#16#FBC2; (* < 64450 - DCDC3LL *)
    PGN_DC_DC_CONVERTER_3_HIGH_SIDE_LIMITS : UDINT := UDINT#16#FBC3; (* < 64451 - DCDC3HL *)
    PGN_DC_DC_CONVERTER_2_LIFETIME_DATA : UDINT := UDINT#16#FBC4; (* < 64452 - DCDC2LD *)
    PGN_DC_DC_CONVERTER_2_CONFIGURATION_1 : UDINT := UDINT#16#FBC5; (* < 64453 - DCDC2CFG1 *)
    PGN_DC_DC_CONVERTER_2_SLI_BATTERY_LIMITS : UDINT := UDINT#16#FBC6; (* < 64454 - DCDC2SBL *)
    PGN_DC_DC_CONVERTER_2_TEMPERATURES : UDINT := UDINT#16#FBC7; (* < 64455 - DCDC2T *)
    PGN_DC_DC_CONVERTER_2_LOW_SIDE_LIMITS : UDINT := UDINT#16#FBC8; (* < 64456 - DCDC2LL *)
    PGN_DC_DC_CONVERTER_2_HIGH_SIDE_LIMITS : UDINT := UDINT#16#FBC9; (* < 64457 - DCDC2HL *)
    PGN_CIA_602_2_AUTOSAR_CAN_NM_OBSOLETE : UDINT := UDINT#16#FBCA; (* < 64458 - CACN *)
    PGN_ENGINE_EXHAUST_PARTICULATE_CONTROL_SYSTEM_INFO : UDINT := UDINT#16#FBCB; (* < 64459 - EEPCSI *)
    PGN_WELL_STIMULATION_PUMP_HOURS : UDINT := UDINT#16#FBCC; (* < 64460 - WSPH *)
    PGN_WELL_STIMULATION_PUMP_SYSTEM_CONFIGURATION_STATUS : UDINT := UDINT#16#FBCD; (* < 64461 - WSPT2 *)
    PGN_CONFIGURABLE_RECEIVE_SPNS_STATUS : UDINT := UDINT#16#FBCE; (* < 64462 - CRSS *)
    PGN_DC_DC_CONVERTER_1_LIFETIME_DATA : UDINT := UDINT#16#FBCF; (* < 64463 - DCDC1LD *)
    PGN_DC_DC_CONVERTER_1_CONFIGURATION_1 : UDINT := UDINT#16#FBD0; (* < 64464 - DCDC1CFG1 *)
    PGN_DC_DC_CONVERTER_1_SLI_BATTERY_LIMITS : UDINT := UDINT#16#FBD1; (* < 64465 - DCDC1SBL *)
    PGN_PUMP_OIL_MESSAGE : UDINT := UDINT#16#FBD2; (* < 64466 - POM *)
    PGN_WELL_STIMULATION_PUMP_SYSTEM_LIFETIME_TOTALS : UDINT := UDINT#16#FBD3; (* < 64467 - WSPT *)
    PGN_WELL_STIMULATION_PUMP_SYSTEM_CONFIGURATION : UDINT := UDINT#16#FBD4; (* < 64468 - WSPC *)
    PGN_AFTERCOOLER_AND_OIL_COOLER_FLUIDS_2 : UDINT := UDINT#16#FBD5; (* < 64469 - ACOCF2 *)
    PGN_ELECTRONIC_ENGINE_CONTROLLER_21 : UDINT := UDINT#16#FBD6; (* < 64470 - EEC21 *)
    PGN_CONFIGURABLE_TRANSMIT_PGNS_STATUS : UDINT := UDINT#16#FBD7; (* < 64471 - CTPS *)
    PGN_DC_DC_CONVERTER_1_TEMPERATURES : UDINT := UDINT#16#FBD8; (* < 64472 - DCDC1T *)
    PGN_DC_DC_CONVERTER_1_LOW_SIDE_LIMITS : UDINT := UDINT#16#FBD9; (* < 64473 - DCDC1LL *)
    PGN_DC_DC_CONVERTER_1_HIGH_SIDE_LIMITS : UDINT := UDINT#16#FBDA; (* < 64474 - DCDC1HL *)
    PGN_RESERVED_FOR_DIAGNOSTIC_MESSAGE : UDINT := UDINT#16#FBDB; (* < 64475 - DM58 *)
    PGN_DOOR_CONTROL_4 : UDINT := UDINT#16#FBDC; (* < 64476 - DC4 *)
    PGN_DOOR_CONTROL_3 : UDINT := UDINT#16#FBDD; (* < 64477 - DC3 *)
    PGN_ENGINE_TEMPERATURE_6 : UDINT := UDINT#16#FBDE; (* < 64478 - ET6 *)
    PGN_INTAKE_EXHAUST_CONDITIONS_3 : UDINT := UDINT#16#FBDF; (* < 64479 - IC3 *)
    PGN_AFTERCOOLER_AND_OIL_COOLER_FLUIDS_1 : UDINT := UDINT#16#FBE0; (* < 64480 - ACOCF1 *)
    PGN_DIODE_TEMPERATURE_2 : UDINT := UDINT#16#FBE1; (* < 64481 - DT2 *)
    PGN_DIODE_TEMPERATURE_1 : UDINT := UDINT#16#FBE2; (* < 64482 - DT1 *)
    PGN_ALTERNATOR_TEMPERATURE_2 : UDINT := UDINT#16#FBE3; (* < 64483 - AT2 *)
    PGN_FUEL_INFORMATION_7_GASEOUS : UDINT := UDINT#16#FBE4; (* < 64484 - GFI7 *)
    PGN_HIGH_VOLTAGE_ENERGY_STORAGE_SYSTEM_FAN_STATUS_1 : UDINT := UDINT#16#FBE5; (* < 64485 - HVESSFS1 *)
    PGN_HIGH_VOLTAGE_ENERGY_STORAGE_SYSTEM_FAN_COMMANDS : UDINT := UDINT#16#FBE6; (* < 64486 - HVESSFC *)
    PGN_SCR_OPERATOR_INDUCEMENT_INFORMATION_5 : UDINT := UDINT#16#FBE7; (* < 64487 - SCROII5 *)
    PGN_AFTERTREATMENT_SYSTEM_INFORMATION_2 : UDINT := UDINT#16#FBE8; (* < 64488 - ASI2 *)
    PGN_ETHERNET_1_CONNECTION_INFORMATION_2 : UDINT := UDINT#16#FBE9; (* < 64489 - E1NET2 *)
    PGN_ETHERNET_1_CONNECTION_INFORMATION_1 : UDINT := UDINT#16#FBEA; (* < 64490 - E1NET1 *)
    PGN_OIL_DEBRIS_MONITOR_COUNTS_FERROUS_BINS_1_2 : UDINT := UDINT#16#FBEB; (* < 64491 - ODMCF1_2 *)
    PGN_OIL_DEBRIS_MONITOR_COUNTS_FERROUS_BINS_3_4 : UDINT := UDINT#16#FBEC; (* < 64492 - ODMCF3_4 *)
    PGN_OIL_DEBRIS_MONITOR_COUNTS_FERROUS_BINS_5_6 : UDINT := UDINT#16#FBED; (* < 64493 - ODMCF5_6 *)
    PGN_OIL_DEBRIS_MONITOR_COUNTS_NON_FERROUS_BINS_1_2 : UDINT := UDINT#16#FBEE; (* < 64494 - ODMCNF1_2 *)
    PGN_OIL_DEBRIS_MONITOR_COUNTS_NON_FERROUS_BINS_3_4 : UDINT := UDINT#16#FBEF; (* < 64495 - ODMCNF3_4 *)
    PGN_OIL_DEBRIS_MONITOR_COUNTS_NON_FERROUS_BINS_5_6 : UDINT := UDINT#16#FBF0; (* < 64496 - ODMCNF5_6 *)
    PGN_OIL_DEBRIS_MONITORING_SYSTEM_STATUS : UDINT := UDINT#16#FBF1; (* < 64497 - ODMSS *)
    PGN_ENGINE_FUEL_LUBE_SYSTEMS_3 : UDINT := UDINT#16#FBF2; (* < 64498 - EFS3 *)
    PGN_CRUISE_CONTROL_VEHICLE_SPEED_5 : UDINT := UDINT#16#FBF3; (* < 64499 - CCVS5 *)
    PGN_AFTERTREATMENT_2_DIESEL_OXIDATION_CATALYST_2 : UDINT := UDINT#16#FBF4; (* < 64500 - A2DOC2 *)
    PGN_AFTERTREATMENT_1_DIESEL_OXIDATION_CATALYST_2 : UDINT := UDINT#16#FBF5; (* < 64501 - A1DOC2 *)
    PGN_VEHICLE_POSITION_2 : UDINT := UDINT#16#FBF6; (* < 64502 - VP2 *)
    PGN_ELECTRIFIED_ACCESSORY_PROPULSION_MOTOR_COOLANT_FAN_3_STATUS_1 : UDINT := UDINT#16#FBF7; (* < 64503 - EAPMCF3S1 *)
    PGN_ELECTRIFIED_ACCESSORY_PROPULSION_MOTOR_COOLANT_FAN_2_STATUS_1 : UDINT := UDINT#16#FBF8; (* < 64504 - EAPMCF2S1 *)
    PGN_ELECTRIFIED_ACCESSORY_PROPULSION_MOTOR_COOLANT_FAN_1_STATUS_1 : UDINT := UDINT#16#FBF9; (* < 64505 - EAPMCF1S1 *)
    PGN_ELECTRIFIED_ACCESSORY_POWER_ELECTRONICS_COOLANT_FAN_3_STATUS_1 : UDINT := UDINT#16#FBFA; (* < 64506 - EAPECF3S1 *)
    PGN_ELECTRIFIED_ACCESSORY_POWER_ELECTRONICS_COOLANT_FAN_2_STATUS_1 : UDINT := UDINT#16#FBFB; (* < 64507 - EAPECF2S1 *)
    PGN_ELECTRIFIED_ACCESSORY_POWER_ELECTRONICS_COOLANT_FAN_1_STATUS_1 : UDINT := UDINT#16#FBFC; (* < 64508 - EAPECF1S1 *)
    PGN_ELECTRIFIED_ACCESSORY_PROPULSION_MOTOR_OIL_PUMP_STATUS_1 : UDINT := UDINT#16#FBFD; (* < 64509 - EAPMOPS1 *)
    PGN_ELECTRIFIED_ACCESSORY_PROPULSION_MOTOR_COOLANT_PUMP_STATUS_1 : UDINT := UDINT#16#FBFE; (* < 64510 - EAPMCPS1 *)
    PGN_ELECTRIFIED_ACCESSORY_POWER_ELECTRONICS_COOLANT_PUMP_STATUS_1 : UDINT := UDINT#16#FBFF; (* < 64511 - EAPECPS1 *)
    PGN_TRAILER_WHEEL_BRAKE_WEAR_LIFE_REMAINING_INFORMATION : UDINT := UDINT#16#FC00; (* < 64512 - TWBW *)
    PGN_ELECTRIFIED_ACCESSORY_MOTOR_STATUS_1 : UDINT := UDINT#16#FC01; (* < 64513 - EAMS1 *)
    PGN_SCR_SYSTEM_INFORMATION : UDINT := UDINT#16#FC02; (* < 64514 - SCRSI *)
    PGN_VEHICLE_ELECTRICAL_POWER_14 : UDINT := UDINT#16#FC03; (* < 64515 - VEP14 *)
    PGN_VEHICLE_ELECTRICAL_POWER_13 : UDINT := UDINT#16#FC04; (* < 64516 - VEP13 *)
    PGN_VEHICLE_ELECTRICAL_POWER_12 : UDINT := UDINT#16#FC05; (* < 64517 - VEP12 *)
    PGN_VEHICLE_ELECTRICAL_POWER_11 : UDINT := UDINT#16#FC06; (* < 64518 - VEP11 *)
    PGN_VEHICLE_ELECTRICAL_POWER_10 : UDINT := UDINT#16#FC07; (* < 64519 - VEP10 *)
    PGN_VEHICLE_ELECTRICAL_POWER_9 : UDINT := UDINT#16#FC08; (* < 64520 - VEP9 *)
    PGN_VEHICLE_ELECTRICAL_POWER_8 : UDINT := UDINT#16#FC09; (* < 64521 - VEP8 *)
    PGN_VEHICLE_ELECTRICAL_POWER_7 : UDINT := UDINT#16#FC0A; (* < 64522 - VEP7 *)
    PGN_ELECTRONIC_ENGINE_CONTROLLER_20 : UDINT := UDINT#16#FC0B; (* < 64523 - EEC20 *)
    PGN_EVAPORATIVE_SYSTEMS : UDINT := UDINT#16#FC0C; (* < 64524 - EVAP *)
    PGN_FIRE_PUMP_STATISTICS_1 : UDINT := UDINT#16#FC0D; (* < 64525 - FPS1 *)
    PGN_PRIMARY_OR_REAR_HITCH_ROLL_AND_PITCH_SENSITIVITY : UDINT := UDINT#16#FC0E; (* < 64526 - PHRPS *)
    PGN_SECONDARY_OR_FRONT_HITCH_ROLL_AND_PITCH_SENSITIVITY : UDINT := UDINT#16#FC0F; (* < 64527 - SHRPS *)
    PGN_AMBIENT_CONDITIONS_3 : UDINT := UDINT#16#FC10; (* < 64528 - AMB3 *)
    PGN_TOTAL_GASEOUS_FUEL_INFORMATION : UDINT := UDINT#16#FC11; (* < 64529 - TGFI *)
    PGN_CAB_DOOR_CONTROL_1 : UDINT := UDINT#16#FC12; (* < 64530 - CDC1 *)
    PGN_DOOR_LATCH_STATUS : UDINT := UDINT#16#FC13; (* < 64531 - DLS *)
    PGN_VEHICLE_ELECTRICAL_POWER_3_OBSOLETE_USE_PGN_65106 : UDINT := UDINT#16#FC14; (* < 64532 - Vehicle Electrical Power 3 (obsolete, use PGN 65106) *)
    PGN_VEHICLE_ELECTRICAL_POWER_6 : UDINT := UDINT#16#FC15; (* < 64533 - VEP6 *)
    PGN_PAYLOAD_TEMPERATURE_2 : UDINT := UDINT#16#FC16; (* < 64534 - PLT2 *)
    PGN_PAYLOAD_TEMPERATURE_1 : UDINT := UDINT#16#FC17; (* < 64535 - PLT1 *)
    PGN_PAYLOAD_SYSTEM_TOTALS_2 : UDINT := UDINT#16#FC18; (* < 64536 - PLST2 *)
    PGN_PAYLOAD_SYSTEM_TOTALS_1 : UDINT := UDINT#16#FC19; (* < 64537 - PLST1 *)
    PGN_HVESS_THERMAL_MANAGEMENT_SYSTEM_CONTROL_1 : UDINT := UDINT#16#FC1A; (* < 64538 - HVESSTC1 *)
    PGN_HVESS_THERMAL_MANAGEMENT_SYSTEM_CONTROL_2 : UDINT := UDINT#16#FC1B; (* < 64539 - HVESSTC2 *)
    PGN_REFRIGERATION_COMPARTMENT_INFORMATION_1 : UDINT := UDINT#16#FC1C; (* < 64540 - RCI1 *)
    PGN_REFRIGERATION_COMPARTMENT_INFORMATION_2 : UDINT := UDINT#16#FC1D; (* < 64541 - RCI2 *)
    PGN_VEHICLE_ELECTRICAL_POWER_16 : UDINT := UDINT#16#FC1E; (* < 64542 - VEP16 *)
    PGN_VEHICLE_ELECTRICAL_POWER_17 : UDINT := UDINT#16#FC1F; (* < 64543 - VEP17 *)
    PGN_HIGH_VOLTAGE_ENERGY_STORAGE_SYSTEM_MODULE_STATUS_2 : UDINT := UDINT#16#FC20; (* < 64544 - HVESSMS2 *)
    PGN_HIGH_VOLTAGE_ENERGY_STORAGE_SYSTEM_MODULE_STATUS_3 : UDINT := UDINT#16#FC21; (* < 64545 - HVESSMS3 *)
    PGN_ELECTRONIC_ENGINE_CONTROLLER_19 : UDINT := UDINT#16#FC22; (* < 64546 - EEC19 *)
    PGN_FUEL_CONSUMPTION_LIQUID_2 : UDINT := UDINT#16#FC23; (* < 64547 - LFC2 *)
    PGN_AFTERTREATMENT_2_DIESEL_EXHAUST_FLUID_TANK_1_INFORMATION_2 : UDINT := UDINT#16#FC24; (* < 64548 - AT2T1I2 *)
    PGN_AFTERTREATMENT_1_DIESEL_EXHAUST_FLUID_TANK_1_INFORMATION_2 : UDINT := UDINT#16#FC25; (* < 64549 - AT1T1I2 *)
    PGN_AFTERTREATMENT_2_DIESEL_EXHAUST_FLUID_INFORMATION_2 : UDINT := UDINT#16#FC26; (* < 64550 - A2DEFI2 *)
    PGN_AFTERTREATMENT_1_DIESEL_EXHAUST_FLUID_INFORMATION_2 : UDINT := UDINT#16#FC27; (* < 64551 - A1DEFI2 *)
    PGN_CRUISE_CONTROL_VEHICLE_SPEED_6 : UDINT := UDINT#16#FC28; (* < 64552 - CCVS6 *)
    PGN_FORWARD_LANE_IMAGE_3 : UDINT := UDINT#16#FC29; (* < 64553 - FLI3 *)
    PGN_OPERATOR_INDUCEMENT_INFORMATION_1 : UDINT := UDINT#16#FC2A; (* < 64554 - OII1 *)
    PGN_CRUISE_CONTROL_VEHICLE_SPEED_4 : UDINT := UDINT#16#FC2B; (* < 64555 - CCVS4 *)
    PGN_BRAKE_CALIPER_LINING_CLEARANCE : UDINT := UDINT#16#FC2C; (* < 64556 - BCLC *)
    PGN_ALTERNATE_FUEL_5 : UDINT := UDINT#16#FC2D; (* < 64557 - AF5 *)
    PGN_ENGINE_TURBOCHARGER_CONTROL_3 : UDINT := UDINT#16#FC2E; (* < 64558 - ETCC3 *)
    PGN_FIRE_SUPPRESSION_AGENT_STATUS : UDINT := UDINT#16#FC2F; (* < 64559 - FSAS *)
    PGN_SCR_OPERATOR_INDUCEMENT_INFORMATION_4 : UDINT := UDINT#16#FC30; (* < 64560 - SCROII4 *)
    PGN_AFTERTREATMENT_SYSTEM_INFORMATION_1 : UDINT := UDINT#16#FC31; (* < 64561 - ASI1 *)
    PGN_AFTERTREATMENT_1_PARTICULATE_SENSOR_INFORMATION_3 : UDINT := UDINT#16#FC32; (* < 64562 - AFT1PSI3 *)
    PGN_ENGINE_FUEL_INJECTOR_METERING_RAIL_PRESSURE_INFORMATION_3 : UDINT := UDINT#16#FC33; (* < 64563 - EFIMRPI3 *)
    PGN_ENGINE_FUEL_INJECTOR_METERING_RAIL_PRESSURE_INFORMATION_2 : UDINT := UDINT#16#FC34; (* < 64564 - EFIMRPI2 *)
    PGN_AFTERTREATMENT_2_DIESEL_EXHAUST_FLUID_PUMP_1_INFORMATION : UDINT := UDINT#16#FC35; (* < 64565 - AT2P1I *)
    PGN_GASEOUS_FUEL_SUPPLY_VALVE_INFORMATION : UDINT := UDINT#16#FC36; (* < 64566 - GFSVI *)
    PGN_ENGINE_OIL_MIST_DETECTION_INFORMATION_2 : UDINT := UDINT#16#FC37; (* < 64567 - EOMDI2 *)
    PGN_ENGINE_OIL_MIST_DETECTION_INFORMATION_1 : UDINT := UDINT#16#FC38; (* < 64568 - EOMDI1 *)
    PGN_GASEOUS_FUEL_SUPPLY_PRESSURE_2 : UDINT := UDINT#16#FC39; (* < 64569 - GFSP2 *)
    PGN_GASEOUS_FUEL_SUPPLY_PRESSURE_1 : UDINT := UDINT#16#FC3A; (* < 64570 - GFSP1 *)
    PGN_ENGINE_END_BEARING_TEMPERATURE_3 : UDINT := UDINT#16#FC3B; (* < 64571 - EEBT3 *)
    PGN_ENGINE_END_BEARING_TEMPERATURE_2 : UDINT := UDINT#16#FC3C; (* < 64572 - EEBT2 *)
    PGN_ENGINE_END_BEARING_TEMPERATURE_1 : UDINT := UDINT#16#FC3D; (* < 64573 - EEBT1 *)
    PGN_HEAT_EXCHANGER_DEBRIS_PURGE_INFORMATION : UDINT := UDINT#16#FC3E; (* < 64574 - HEDPI *)
    PGN_ENGINE_TURBOCHARGER_CONTROL_2 : UDINT := UDINT#16#FC3F; (* < 64575 - ETCC2 *)
    PGN_ENGINE_HYDRAULIC_FUEL_2_PUMP_STATUS : UDINT := UDINT#16#FC40; (* < 64576 - EHF2PC *)
    PGN_ALTERNATE_FUEL_4 : UDINT := UDINT#16#FC41; (* < 64577 - AF4 *)
    PGN_TIRE_CONDITION_MESSAGE_2 : UDINT := UDINT#16#FC42; (* < 64578 - TIRE2 *)
    PGN_TIRE_CONFIGURATION_STATUS_INFORMATION : UDINT := UDINT#16#FC43; (* < 64579 - TCSI *)
    PGN_HIGH_VOLTAGE_ENERGY_STORAGE_SYSTEM_DATA_15 : UDINT := UDINT#16#FC44; (* < 64580 - HVESSD15 *)
    PGN_TIRE_WIRELESS_SIGNAL_STRENGTH_INDICATOR : UDINT := UDINT#16#FC45; (* < 64581 - TWSSI *)
    PGN_TIRE_SENSOR_IDENTIFICATION_STATUS : UDINT := UDINT#16#FC46; (* < 64582 - TSIS *)
    PGN_MONITORED_TIRE_INFORMATION : UDINT := UDINT#16#FC47; (* < 64583 - MTI *)
    PGN_AFTERTREATMENT_2_HISTORICAL_INFORMATION_2 : UDINT := UDINT#16#FC48; (* < 64584 - AT2HI2 *)
    PGN_AFTERTREATMENT_1_HISTORICAL_INFORMATION_2 : UDINT := UDINT#16#FC49; (* < 64585 - AT1HI2 *)
    PGN_SCR_SYSTEM_CLEANING : UDINT := UDINT#16#FC4A; (* < 64586 - SCRSC *)
    PGN_ELECTRONIC_ENGINE_CONTROLLER_17 : UDINT := UDINT#16#FC4B; (* < 64587 - EEC17 *)
    PGN_SCR_OPERATOR_INDUCEMENT_INFORMATION_3 : UDINT := UDINT#16#FC4C; (* < 64588 - SCROII3 *)
    PGN_AFTERTREATMENT_2_SCR_DOSING_SYSTEM_INFORMATION_3 : UDINT := UDINT#16#FC4D; (* < 64589 - A2SCRDSI3 *)
    PGN_AFTERTREATMENT_1_SCR_DOSING_SYSTEM_INFORMATION_3 : UDINT := UDINT#16#FC4E; (* < 64590 - A1SCRDSI3 *)
    PGN_PAYLOAD_WEIGHT_SENSOR_INFORMATION : UDINT := UDINT#16#FC4F; (* < 64591 - PWSI *)
    PGN_PAYLOAD_SYSTEM_STATUS : UDINT := UDINT#16#FC50; (* < 64592 - PLSS *)
    PGN_AIR_SUSPENSION_CONTROL_7 : UDINT := UDINT#16#FC51; (* < 64593 - ASC7 *)
    PGN_BIN_WEIGHT_AND_LIFT_COUNT : UDINT := UDINT#16#FC52; (* < 64594 - BWLN *)
    PGN_ENGINE_GASEOUS_LEAKAGE_INFORMATION : UDINT := UDINT#16#FC53; (* < 64595 - EGLI *)
    PGN_DRIVING_AND_REST_TIMES_DRIVER_2 : UDINT := UDINT#16#FC54; (* < 64596 - DTR2 *)
    PGN_DRIVING_AND_REST_TIMES_DRIVER_1 : UDINT := UDINT#16#FC55; (* < 64597 - DTR1 *)
    PGN_SCR_OPERATOR_INDUCEMENT_INFORMATION_2 : UDINT := UDINT#16#FC56; (* < 64598 - SCROII2 *)
    PGN_SCR_OPERATOR_INDUCEMENT_INFORMATION_1 : UDINT := UDINT#16#FC57; (* < 64599 - SCROII1 *)
    PGN_TURBOCHARGER_INFORMATION_7 : UDINT := UDINT#16#FC58; (* < 64600 - TCI7 *)
    PGN_ENGINE_LOAD_SHARING_INFORMATION : UDINT := UDINT#16#FC59; (* < 64601 - ELS *)
    PGN_SYNCHRONIZED_SERVICE_DISTANCE_INFORMATION : UDINT := UDINT#16#FC5A; (* < 64602 - SSDI *)
    PGN_SYNCHRONIZED_SERVICE_DELAY_OPERATIONAL_TIME_BASED_INFORMATION : UDINT := UDINT#16#FC5B; (* < 64603 - SSOTI *)
    PGN_SYNCHRONIZED_SERVICE_DELAY_CALENDAR_TIME_BASED_INFORMATION : UDINT := UDINT#16#FC5C; (* < 64604 - SSCTI *)
    PGN_HIGH_VOLTAGE_ENERGY_STORAGE_SYSTEM_CONFIGURATION : UDINT := UDINT#16#FC5D; (* < 64605 - HVESSCFG *)
    PGN_HIGH_VOLTAGE_ENERGY_STORAGE_SYSTEM_HISTORY : UDINT := UDINT#16#FC5E; (* < 64606 - HVESSHIST *)
    PGN_ENCODER_POSITION : UDINT := UDINT#16#FC5F; (* < 64607 - EPOS *)
    PGN_ENCODER_HIGH_RESOLUTION_POSITION : UDINT := UDINT#16#FC60; (* < 64608 - EHRPOS *)
    PGN_ENCODER_SPEED : UDINT := UDINT#16#FC61; (* < 64609 - ESPD *)
    PGN_ENCODER_ACCELERATION : UDINT := UDINT#16#FC62; (* < 64610 - EACC *)
    PGN_ENCODER_POSITION_WITH_SPEED_AND_ACCELERATION : UDINT := UDINT#16#FC63; (* < 64611 - EPSAC *)
    PGN_INCLINOMETER_SLOPE_LONGITUDINAL_16_BIT : UDINT := UDINT#16#FC64; (* < 64612 - ISLONG16 *)
    PGN_INCLINOMETER_SLOPE_LONGITUDINAL_32_BIT : UDINT := UDINT#16#FC65; (* < 64613 - ISLONG32 *)
    PGN_INCLINOMETER_SLOPE_LATERAL_16_BIT : UDINT := UDINT#16#FC66; (* < 64614 - ISLAT16 *)
    PGN_INCLINOMETER_SLOPE_LATERAL_32_BIT : UDINT := UDINT#16#FC67; (* < 64615 - ISLAT32 *)
    PGN_CANOPEN_EMERGENCY_MESSAGE : UDINT := UDINT#16#FC68; (* < 64616 - CEM *)
    PGN_EV_OPERATOR_INDICATORS_1 : UDINT := UDINT#16#FC69; (* < 64617 - EVOI1 *)
    PGN_SYSTEM_IDENTIFICATION : UDINT := UDINT#16#FC6A; (* < 64618 - SYSTEMID *)
    PGN_ENGINE_MAXIMUM_NET_TORQUE_MAP_OBSOLETE_USE_PGN_64248 : UDINT := UDINT#16#FC6B; (* < 64619 - Engine Maximum Net Torque Map (obsolete, use PGN 64248) *)
    PGN_ALARM : UDINT := UDINT#16#FC6C; (* < 64620 - ALARM *)
    PGN_ACOUSTIC_WARNING_REQUEST : UDINT := UDINT#16#FC6D; (* < 64621 - AWR *)
    PGN_ACOUSTIC_WARNING_STATE : UDINT := UDINT#16#FC6E; (* < 64622 - AWS *)
    PGN_VEHICLE_LOAD : UDINT := UDINT#16#FC6F; (* < 64623 - AXL *)
    PGN_BODY_APPLICATION_UNIT_1 : UDINT := UDINT#16#FC70; (* < 64624 - BAU1 *)
    PGN_BODY_APPLICATION_UNIT_2 : UDINT := UDINT#16#FC71; (* < 64625 - BAU2 *)
    PGN_BODY_APPLICATION_UNIT_3 : UDINT := UDINT#16#FC72; (* < 64626 - BAU3 *)
    PGN_BODY_APPLICATION_UNIT_4 : UDINT := UDINT#16#FC73; (* < 64627 - BAU4 *)
    PGN_BODY_APPLICATION_UNIT_5 : UDINT := UDINT#16#FC74; (* < 64628 - BAU5 *)
    PGN_BODY_APPLICATION_UNIT_6 : UDINT := UDINT#16#FC75; (* < 64629 - BAU6 *)
    PGN_BODY_APPLICATION_UNIT_7 : UDINT := UDINT#16#FC76; (* < 64630 - BAU7 *)
    PGN_BODY_APPLICATION_UNIT_8 : UDINT := UDINT#16#FC77; (* < 64631 - BAU8 *)
    PGN_ELECTRONIC_CONTROL_UNIT : UDINT := UDINT#16#FC78; (* < 64632 - ECU *)
    PGN_ECU_POWER_SUPPLY : UDINT := UDINT#16#FC79; (* < 64633 - ECU_PWR *)
    PGN_ECU_TEMPERATURE : UDINT := UDINT#16#FC7A; (* < 64634 - ECU_TMP *)
    PGN_ERROR : UDINT := UDINT#16#FC7B; (* < 64635 - ERROR *)
    PGN_HEATING_AND_REFRIGERATING_UNIT_1 : UDINT := UDINT#16#FC7C; (* < 64636 - HRU1 *)
    PGN_HEATING_AND_REFRIGERATING_UNIT_2 : UDINT := UDINT#16#FC7D; (* < 64637 - HRU2 *)
    PGN_HEATING_AND_REFRIGERATING_UNIT_3 : UDINT := UDINT#16#FC7E; (* < 64638 - HRU3 *)
    PGN_HEATING_AND_REFRIGERATING_UNIT_4 : UDINT := UDINT#16#FC7F; (* < 64639 - HRU4 *)
    PGN_HRU_TEMPERATURE_SETPOINT : UDINT := UDINT#16#FC80; (* < 64640 - HTS *)
    PGN_LIFTING_UNIT_1 : UDINT := UDINT#16#FC81; (* < 64641 - LU1 *)
    PGN_TAIL_LIFT_UNIT_1 : UDINT := UDINT#16#FC82; (* < 64642 - TLU1 *)
    PGN_VEHICLE_STATUS : UDINT := UDINT#16#FC83; (* < 64643 - VS *)
    PGN_WINDSHIELD_WIPER_REQUEST : UDINT := UDINT#16#FC84; (* < 64644 - WWR *)
    PGN_FUEL_CELL_AUXILIARY_HEATER_CONTROL : UDINT := UDINT#16#FC85; (* < 64645 - FCHTRC *)
    PGN_FUEL_CELL_AUXILIARY_HEATER_INFORMATION : UDINT := UDINT#16#FC86; (* < 64646 - FCHTR *)
    PGN_FUEL_CELL_COOLANT_PUMP_1_COMMAND : UDINT := UDINT#16#FC87; (* < 64647 - FCCP1C *)
    PGN_FUEL_CELL_COOLANT_PUMP_2_COMMAND : UDINT := UDINT#16#FC88; (* < 64648 - FCCP2C *)
    PGN_FUEL_CELL_COOLANT_PUMP_1_STATUS : UDINT := UDINT#16#FC89; (* < 64649 - FCCP1S *)
    PGN_FUEL_CELL_COOLANT_PUMP_2_STATUS : UDINT := UDINT#16#FC8A; (* < 64650 - FCCP2S *)
    PGN_AFTERTREATMENT_1_PARTICULATE_SENSOR_INFORMATION_2 : UDINT := UDINT#16#FC8B; (* < 64651 - AFT1PSI2 *)
    PGN_AFTERTREATMENT_1_PARTICULATE_SENSOR_INFORMATION_1 : UDINT := UDINT#16#FC8C; (* < 64652 - AFT1PSI1 *)
    PGN_PRODUCT_IDENTIFICATION : UDINT := UDINT#16#FC8D; (* < 64653 - PII *)
    PGN_FUNCTIONALI_CHARACTERISTICS : UDINT := UDINT#16#FC8E; (* < 64654 - CFF *)
    PGN_ALTERNATE_FUEL_3 : UDINT := UDINT#16#FC8F; (* < 64655 - AF3 *)
    PGN_ENGINE_FUEL_INJECTOR_METERING_RAIL_PRESSURE_INFORMATION_1 : UDINT := UDINT#16#FC90; (* < 64656 - EFIMRPI1 *)
    PGN_ENGINE_EXHAUST_NOX : UDINT := UDINT#16#FC91; (* < 64657 - EEN *)
    PGN_AIR_FUEL_RATIO_1 : UDINT := UDINT#16#FC92; (* < 64658 - AFR1 *)
    PGN_GASEOUS_FUEL_PRESSURE_2 : UDINT := UDINT#16#FC93; (* < 64659 - GFP2 *)
    PGN_AFTERTREATMENT_SYSTEM_ABUSE_INFORMATION : UDINT := UDINT#16#FC94; (* < 64660 - ASAI *)
    PGN_ENGINE_CYLINDER_PRESSURE_MONITOR_STATUS_INFORMATION : UDINT := UDINT#16#FC95; (* < 64661 - ECPMSI *)
    PGN_ENGINE_INFORMATION_2 : UDINT := UDINT#16#FC96; (* < 64662 - EI2 *)
    PGN_ELECTRONIC_STEERING_CONTROL_2 : UDINT := UDINT#16#FC97; (* < 64663 - ESC2 *)
    PGN_VEHICLE_SPEED_LIMITER : UDINT := UDINT#16#FC98; (* < 64664 - VSL *)
    PGN_ASSEMBLY_UNIT_IDENTIFICATION : UDINT := UDINT#16#FC99; (* < 64665 - AUI *)
    PGN_JOYSTICK_3_LAMP_STATUS : UDINT := UDINT#16#FC9A; (* < 64666 - JS3LS *)
    PGN_JOYSTICK_2_LAMP_STATUS : UDINT := UDINT#16#FC9B; (* < 64667 - JS2LS *)
    PGN_JOYSTICK_1_LAMP_STATUS : UDINT := UDINT#16#FC9C; (* < 64668 - JS1LS *)
    PGN_ENGINE_TIMING_ACTUATOR_POSITION_COMMAND : UDINT := UDINT#16#FC9D; (* < 64669 - ETAPC *)
    PGN_ENGINE_TIMING_ACTUATOR_POSITION : UDINT := UDINT#16#FC9E; (* < 64670 - ETAP *)
    PGN_DASH_DISPLAY_2 : UDINT := UDINT#16#FC9F; (* < 64671 - DD2 *)
    PGN_MULTI_FUEL_ENGINE_HOURS : UDINT := UDINT#16#FCA0; (* < 64672 - MFEH *)
    PGN_ENGINE_SPARK_MISFIRE_RATE_3 : UDINT := UDINT#16#FCA1; (* < 64673 - ESMR3 *)
    PGN_ENGINE_SPARK_MISFIRE_RATE_2 : UDINT := UDINT#16#FCA2; (* < 64674 - ESMR2 *)
    PGN_ENGINE_SPARK_MISFIRE_RATE_1 : UDINT := UDINT#16#FCA3; (* < 64675 - ESMR1 *)
    PGN_ENGINE_SPARK_MAXIMUM_VOLTAGE_6 : UDINT := UDINT#16#FCA4; (* < 64676 - ESVMAX6 *)
    PGN_ENGINE_SPARK_MAXIMUM_VOLTAGE_5 : UDINT := UDINT#16#FCA5; (* < 64677 - ESVMAX5 *)
    PGN_ENGINE_SPARK_MAXIMUM_VOLTAGE_4 : UDINT := UDINT#16#FCA6; (* < 64678 - ESVMAX4 *)
    PGN_ENGINE_SPARK_MAXIMUM_VOLTAGE_3 : UDINT := UDINT#16#FCA7; (* < 64679 - ESVMAX3 *)
    PGN_ENGINE_SPARK_MAXIMUM_VOLTAGE_2 : UDINT := UDINT#16#FCA8; (* < 64680 - ESVMAX2 *)
    PGN_ENGINE_SPARK_MAXIMUM_VOLTAGE_1 : UDINT := UDINT#16#FCA9; (* < 64681 - ESVMAX1 *)
    PGN_ENGINE_SPARK_MINIMUM_VOLTAGE_6 : UDINT := UDINT#16#FCAA; (* < 64682 - ESVMIN6 *)
    PGN_ENGINE_SPARK_MINIMUM_VOLTAGE_5 : UDINT := UDINT#16#FCAB; (* < 64683 - ESVMIN5 *)
    PGN_ENGINE_SPARK_MINIMUM_VOLTAGE_4 : UDINT := UDINT#16#FCAC; (* < 64684 - ESVMIN4 *)
    PGN_ENGINE_SPARK_MINIMUM_VOLTAGE_3 : UDINT := UDINT#16#FCAD; (* < 64685 - ESVMIN3 *)
    PGN_ENGINE_SPARK_MINIMUM_VOLTAGE_2 : UDINT := UDINT#16#FCAE; (* < 64686 - ESVMIN2 *)
    PGN_ENGINE_SPARK_MINIMUM_VOLTAGE_1 : UDINT := UDINT#16#FCAF; (* < 64687 - ESVMIN1 *)
    PGN_ENGINE_IGNITION_CONTROLLER_MAINTENANCE_HOURS : UDINT := UDINT#16#FCB0; (* < 64688 - EICMH *)
    PGN_ENGINE_IGNITION_CONTROL_MODULE_STATUS : UDINT := UDINT#16#FCB1; (* < 64689 - ICMSTS *)
    PGN_SWITCHED_POWER_OUTPUT_CURRENT : UDINT := UDINT#16#FCB2; (* < 64690 - SPOC1 *)
    PGN_FUSED_POWER_OUTPUT_CURRENT : UDINT := UDINT#16#FCB3; (* < 64691 - FPOC *)
    PGN_SWITCHED_POWER_OUTPUT_STATUS : UDINT := UDINT#16#FCB4; (* < 64692 - SPOS *)
    PGN_FUSED_POWER_OUTPUT_STATUS : UDINT := UDINT#16#FCB5; (* < 64693 - FPOS *)
    PGN_VEHICLE_ELECTRICAL_POWER_5 : UDINT := UDINT#16#FCB6; (* < 64694 - VEP5 *)
    PGN_HYBRID_OR_EV_SYSTEM_STATUS_2 : UDINT := UDINT#16#FCB7; (* < 64695 - HSS2 *)
    PGN_AFTERTREATMENT_2_SERVICE_2 : UDINT := UDINT#16#FCB8; (* < 64696 - AT2S2 *)
    PGN_AFTERTREATMENT_1_SERVICE_2 : UDINT := UDINT#16#FCB9; (* < 64697 - AT1S2 *)
    PGN_AFTERTREATMENT_2_SCR_ELECTRONIC_CONTROL_MODULE_INFORMATION : UDINT := UDINT#16#FCBA; (* < 64698 - A2ECMI *)
    PGN_AFTERTREATMENT_1_SCR_ELECTRONIC_CONTROL_MODULE_INFORMATION : UDINT := UDINT#16#FCBB; (* < 64699 - A1ECMI *)
    PGN_AFTERTREATMENT_2_SCR_SERVICE_INFORMATION_2 : UDINT := UDINT#16#FCBC; (* < 64700 - A2SCRSI2 *)
    PGN_AFTERTREATMENT_1_SCR_SERVICE_INFORMATION_2 : UDINT := UDINT#16#FCBD; (* < 64701 - A1SCRSI2 *)
    PGN_ELECTRONIC_TRANSMISSION_CONTROLLER_9 : UDINT := UDINT#16#FCBE; (* < 64702 - ETC9 *)
    PGN_ELECTRONIC_TRANSMISSION_CONTROLLER_10 : UDINT := UDINT#16#FCBF; (* < 64703 - ETC10 *)
    PGN_ELECTRONIC_TRANSMISSION_CONTROLLER_11 : UDINT := UDINT#16#FCC0; (* < 64704 - ETC11 *)
    PGN_TRANSMISSION_FLUIDS_3 : UDINT := UDINT#16#FCC1; (* < 64705 - TRF3 *)
    PGN_HYBRID_OR_EV_SYSTEM_STATUS_1 : UDINT := UDINT#16#FCC2; (* < 64706 - HSS1 *)
    PGN_FUEL_INFORMATION_4_GASEOUS : UDINT := UDINT#16#FCC3; (* < 64707 - GFI4 *)
    PGN_AFTERTREATMENT_2_SCR_EXHAUST_GAS_TEMPERATURE_2 : UDINT := UDINT#16#FCC4; (* < 64708 - A2SCREGT2 *)
    PGN_AFTERTREATMENT_1_SCR_EXHAUST_GAS_TEMPERATURE_2 : UDINT := UDINT#16#FCC5; (* < 64709 - A1SCREGT2 *)
    PGN_OBD_INFORMATION : UDINT := UDINT#16#FCC6; (* < 64710 - DM57 *)
    PGN_MODEL_YEAR_AND_CERTIFICATION_ENGINE_FAMILY : UDINT := UDINT#16#FCC7; (* < 64711 - DM56 *)
    PGN_ELECTRONIC_ENGINE_CONTROLLER_13 : UDINT := UDINT#16#FCC8; (* < 64712 - EEC13 *)
    PGN_ENGINE_FUEL_THROTTLE_VALVE_INFORMATION_2 : UDINT := UDINT#16#FCC9; (* < 64713 - EF/TVI2 *)
    PGN_ENGINE_EXHAUST_GAS_RECIRCULATION_2_ACTUATOR : UDINT := UDINT#16#FCCA; (* < 64714 - EEGR2A *)
    PGN_ENGINE_EXHAUST_GAS_RECIRCULATION_1_ACTUATOR : UDINT := UDINT#16#FCCB; (* < 64715 - EEGR1A *)
    PGN_ELECTRONIC_ENGINE_CONTROLLER_12 : UDINT := UDINT#16#FCCC; (* < 64716 - EEC12 *)
    PGN_DRIVE_STRATEGY_STATUS : UDINT := UDINT#16#FCCD; (* < 64717 - DSS *)
    PGN_DRIVE_STRATEGY_COMMAND : UDINT := UDINT#16#FCCE; (* < 64718 - DSC *)
    PGN_NOX_SENSOR_SELF_DIAGNOSIS_REQUEST : UDINT := UDINT#16#FCCF; (* < 64719 - NSSR *)
    PGN_ENGINE_PARTICULATE_SENSOR_INFORMATION : UDINT := UDINT#16#FCD0; (* < 64720 - EPSI *)
    PGN_ACTIVE_SERVICE_ONLY_DTCS : UDINT := UDINT#16#FCD1; (* < 64721 - DM53 *)
    PGN_PREVIOUSLY_ACTIVE_SERVICE_ONLY_DTCS : UDINT := UDINT#16#FCD2; (* < 64722 - DM54 *)
    PGN_DIAGNOSTIC_DATA_CLEAR_RESET_FOR_ALL_SERVICE_ONLY_DTCS : UDINT := UDINT#16#FCD3; (* < 64723 - DM55 *)
    PGN_XCP_GET_SLAVE_ID : UDINT := UDINT#16#FCD4; (* < 64724 - XCP_ID *)
    PGN_AFTERTREATMENT_1_DIESEL_EXHAUST_FLUID_PUMP_1_INFORMATION : UDINT := UDINT#16#FCD5; (* < 64725 - AT1P1I *)
    PGN_AFTERTREATMENT_1_DIESEL_PARTICULATE_FILTER_2_SOOT_5 : UDINT := UDINT#16#FCD6; (* < 64726 - AT1DPF2S5 *)
    PGN_AFTERTREATMENT_1_DIESEL_PARTICULATE_FILTER_2_SOOT_4 : UDINT := UDINT#16#FCD7; (* < 64727 - AT1DPF2S4 *)
    PGN_AFTERTREATMENT_1_DIESEL_PARTICULATE_FILTER_2_SOOT_3 : UDINT := UDINT#16#FCD8; (* < 64728 - AT1DPF2S3 *)
    PGN_AFTERTREATMENT_1_DIESEL_PARTICULATE_FILTER_1_SOOT_5 : UDINT := UDINT#16#FCD9; (* < 64729 - AT1DPF1S5 *)
    PGN_AFTERTREATMENT_1_DIESEL_PARTICULATE_FILTER_1_SOOT_4 : UDINT := UDINT#16#FCDA; (* < 64730 - AT1DPF1S4 *)
    PGN_AFTERTREATMENT_1_DIESEL_PARTICULATE_FILTER_1_SOOT_3 : UDINT := UDINT#16#FCDB; (* < 64731 - AT1DPF1S3 *)
    PGN_CRUISE_CONTROL_VEHICLE_SPEED_3 : UDINT := UDINT#16#FCDC; (* < 64732 - CCVS3 *)
    PGN_AFTERTREATMENT_2_AIR_CONTROL_3 : UDINT := UDINT#16#FCDD; (* < 64733 - AT2AC3 *)
    PGN_AFTERTREATMENT_1_AIR_CONTROL_3 : UDINT := UDINT#16#FCDE; (* < 64734 - AT1AC3 *)
    PGN_ENGINE_FLUID_LEVEL_PRESSURE_12 : UDINT := UDINT#16#FCDF; (* < 64735 - EFL/P12 *)
    PGN_DIESEL_PARTICULATE_FILTER_CONTROL_2 : UDINT := UDINT#16#FCE0; (* < 64736 - DPFC2 *)
    PGN_FUEL_ECONOMY_2_LIQUID : UDINT := UDINT#16#FCE1; (* < 64737 - LFE2 *)
    PGN_SUPPLEMENTAL_FAN_STATUS : UDINT := UDINT#16#FCE2; (* < 64738 - SFS *)
    PGN_ENGINE_EXHAUST_BRAKE_CONTROL : UDINT := UDINT#16#FCE3; (* < 64739 - EBCC *)
    PGN_ENGINE_FUEL_PROPERTIES : UDINT := UDINT#16#FCE4; (* < 64740 - EFP *)
    PGN_HYDRAULIC_OIL_PROPERTIES : UDINT := UDINT#16#FCE5; (* < 64741 - HOP *)
    PGN_VEHICLE_CHASSIS_LUBRICATION_SYSTEM_2 : UDINT := UDINT#16#FCE6; (* < 64742 - VLS2 *)
    PGN_ENGINE_CONFIGURATION_3 : UDINT := UDINT#16#FCE7; (* < 64743 - EC3 *)
    PGN_INTAKE_VALVE_ACTUATION_CONTROL : UDINT := UDINT#16#FCE8; (* < 64744 - IVAC *)
    PGN_ARMREST_SWITCH_MATRIX_COMMANDS : UDINT := UDINT#16#FCE9; (* < 64745 - ARMSWIMC *)
    PGN_VEHICLE_ELECTRICAL_POWER_4_OBSOLETE_USE_PGN_64695 : UDINT := UDINT#16#FCEA; (* < 64746 - Vehicle Electrical Power 4 (obsolete, use PGN 64695) *)
    PGN_AFTERTREATMENT_2_NOX_ADSORBER_INFORMATION : UDINT := UDINT#16#FCEB; (* < 64747 - AFT2NAI *)
    PGN_AFTERTREATMENT_1_NOX_ADSORBER_INFORMATION : UDINT := UDINT#16#FCEC; (* < 64748 - AFT1NAI *)
    PGN_AFTERTREATMENT_2_WARM_UP_DIESEL_OXIDATION_CATALYST_INFORMATION : UDINT := UDINT#16#FCED; (* < 64749 - AT2WUDOC *)
    PGN_LAND_LEVELING_SYSTEM_REFERENCE_ELEVATION_DATA : UDINT := UDINT#16#FCEE; (* < 64750 - LLRE *)
    PGN_ENGINE_FLUID_LEVEL_PRESSURE_11 : UDINT := UDINT#16#FCEF; (* < 64751 - EFL/P11 *)
    PGN_ENGINE_FUEL_LUBE_SYSTEMS_2 : UDINT := UDINT#16#FCF0; (* < 64752 - EFS2 *)
    PGN_ENGINE_TURBOCHARGER_WASTEGATE_ACTUATOR_AND_EXHAUST_BACK_PRESSURE_REGULATO_X_64753 : UDINT := UDINT#16#FCF1; (* < 64753 - ETWAI1 *)
    PGN_ENGINE_FUEL_THROTTLE_VALVE_INFORMATION_1 : UDINT := UDINT#16#FCF2; (* < 64754 - EFTVI1 *)
    PGN_ENGINE_TURBOCHARGER_COMPRESSOR_BYPASS_INFORMATION : UDINT := UDINT#16#FCF3; (* < 64755 - ETCBI *)
    PGN_CHARGE_AIR_COOLER_2 : UDINT := UDINT#16#FCF4; (* < 64756 - CAC2 *)
    PGN_CHARGE_AIR_COOLER_2_PRECOOLER : UDINT := UDINT#16#FCF5; (* < 64757 - CAC2P *)
    PGN_CHARGE_AIR_COOLER_1 : UDINT := UDINT#16#FCF6; (* < 64758 - CAC1 *)
    PGN_CHARGE_AIR_COOLER_1_PRECOOLER : UDINT := UDINT#16#FCF7; (* < 64759 - CAC1P *)
    PGN_DIESEL_PARTICULATE_FILTER_2_SOOT_2 : UDINT := UDINT#16#FCF8; (* < 64760 - DPF2S2 *)
    PGN_DIESEL_PARTICULATE_FILTER_1_SOOT_2 : UDINT := UDINT#16#FCF9; (* < 64761 - DPF1S2 *)
    PGN_ELECTRONIC_ENGINE_CONTROLLER_11 : UDINT := UDINT#16#FCFA; (* < 64762 - EEC11 *)
    PGN_ENGINE_MANIFOLD_ACTUATOR_POSITION : UDINT := UDINT#16#FCFB; (* < 64763 - EMAP *)
    PGN_ENGINE_MANIFOLD_ACTUATOR_CONTROL : UDINT := UDINT#16#FCFC; (* < 64764 - EMAC *)
    PGN_ELECTRONIC_ENGINE_CONTROLLER_9 : UDINT := UDINT#16#FCFD; (* < 64765 - EEC9 *)
    PGN_ELECTRONIC_ENGINE_CONTROLLER_10 : UDINT := UDINT#16#FCFE; (* < 64766 - EEC10 *)
    PGN_ENGINE_TEMPERATURE_5 : UDINT := UDINT#16#FCFF; (* < 64767 - ET5 *)
    PGN_ENGINE_FLUID_LEVEL_PRESSURE_10 : UDINT := UDINT#16#FD00; (* < 64768 - EFL/P10 *)
    PGN_LOW_VOLTAGE_DISCONNECT_STATUS : UDINT := UDINT#16#FD01; (* < 64769 - LVDS *)
    PGN_STOP_BUTTON : UDINT := UDINT#16#FD02; (* < 64770 - AISO *)
    PGN_IMPLEMENT_OPERATING_STATE : UDINT := UDINT#16#FD03; (* < 64771 - IOS *)
    PGN_DIRECT_LAMP_CONTROL_DATA_2 : UDINT := UDINT#16#FD04; (* < 64772 - DLCD2 *)
    PGN_DIRECT_LAMP_CONTROL_DATA_1 : UDINT := UDINT#16#FD05; (* < 64773 - DLCD1 *)
    PGN_DIRECT_LAMP_CONTROL_COMMAND_2 : UDINT := UDINT#16#FD06; (* < 64774 - DLCC2 *)
    PGN_DIRECT_LAMP_CONTROL_COMMAND_1 : UDINT := UDINT#16#FD07; (* < 64775 - DLCC1 *)
    PGN_ENGINE_OIL_MESSAGE : UDINT := UDINT#16#FD08; (* < 64776 - EOM *)
    PGN_HIGH_RESOLUTION_FUEL_CONSUMPTION_LIQUID : UDINT := UDINT#16#FD09; (* < 64777 - HRLFC *)
    PGN_AFTERTREATMENT_2_OUTLET_GAS_NOX_SENSOR_CORRECTION_DATA_2 : UDINT := UDINT#16#FD0A; (* < 64778 - AT2OGC2 *)
    PGN_AFTERTREATMENT_2_OUTLET_GAS_NOX_SENSOR_CORRECTION_DATA_1 : UDINT := UDINT#16#FD0B; (* < 64779 - AT2OGC1 *)
    PGN_AFTERTREATMENT_2_INTAKE_GAS_NOX_SENSOR_CORRECTION_DATA_2 : UDINT := UDINT#16#FD0C; (* < 64780 - AT2IGC2 *)
    PGN_AFTERTREATMENT_2_INTAKE_GAS_NOX_SENSOR_CORRECTION_DATA_1 : UDINT := UDINT#16#FD0D; (* < 64781 - AT2IGC1 *)
    PGN_AFTERTREATMENT_1_OUTLET_GAS_NOX_SENSOR_CORRECTION_DATA_2 : UDINT := UDINT#16#FD0E; (* < 64782 - AT1OGC2 *)
    PGN_AFTERTREATMENT_1_OUTLET_GAS_NOX_SENSOR_CORRECTION_DATA_1 : UDINT := UDINT#16#FD0F; (* < 64783 - AT1OGC1 *)
    PGN_AFTERTREATMENT_1_INTAKE_GAS_NOX_SENSOR_CORRECTION_DATA_2 : UDINT := UDINT#16#FD10; (* < 64784 - AT1IGC2 *)
    PGN_AFTERTREATMENT_1_INTAKE_GAS_NOX_SENSOR_CORRECTION_DATA_1 : UDINT := UDINT#16#FD11; (* < 64785 - AT1IGC1 *)
    PGN_MAGNET_STATUS_INFORMATION_1 : UDINT := UDINT#16#FD12; (* < 64786 - MSI1 *)
    PGN_MAGNET_SYSTEM_CONFIGURATION_INFORMATION : UDINT := UDINT#16#FD13; (* < 64787 - MSCI *)
    PGN_BATTERY_CHARGER_2 : UDINT := UDINT#16#FD14; (* < 64788 - BCH2 *)
    PGN_BATTERY_CHARGER_1 : UDINT := UDINT#16#FD15; (* < 64789 - BCH1 *)
    PGN_OCCUPANT_CLASSIFICATION_SYSTEM_INFORMATION : UDINT := UDINT#16#FD16; (* < 64790 - OCSI *)
    PGN_BELTLOCK_AND_AIRBAG_DEACTIVATION_SWITCH_INFORMATION : UDINT := UDINT#16#FD17; (* < 64791 - BDS *)
    PGN_COLLISION_SENSOR_INFORMATION : UDINT := UDINT#16#FD18; (* < 64792 - CSI *)
    PGN_IGNITOR_LOOP_INFORMATION : UDINT := UDINT#16#FD19; (* < 64793 - ILI *)
    PGN_AFTERTREATMENT_1_WARM_UP_DIESEL_OXIDATION_CATALYST_INFORMATION : UDINT := UDINT#16#FD1A; (* < 64794 - AT1WUDOC *)
    PGN_DIESEL_PARTICULATE_FILTER_2_SOOT : UDINT := UDINT#16#FD1B; (* < 64795 - DPF2S *)
    PGN_DIESEL_PARTICULATE_FILTER_1_SOOT : UDINT := UDINT#16#FD1C; (* < 64796 - DPF1S *)
    PGN_AFTERTREATMENT_DIFFERENTIAL_TEMPERATURE_2 : UDINT := UDINT#16#FD1D; (* < 64797 - ATDT2 *)
    PGN_AFTERTREATMENT_DIFFERENTIAL_TEMPERATURE_1 : UDINT := UDINT#16#FD1E; (* < 64798 - ATDT1 *)
    PGN_AFTERTREATMENT_2_DIESEL_OXIDATION_CATALYST_1 : UDINT := UDINT#16#FD1F; (* < 64799 - A2DOC1 *)
    PGN_AFTERTREATMENT_1_DIESEL_OXIDATION_CATALYST_1 : UDINT := UDINT#16#FD20; (* < 64800 - A1DOC1 *)
    PGN_AFTERTREATMENT_2_GAS_OXIDATION_CATALYST : UDINT := UDINT#16#FD21; (* < 64801 - A2GOC *)
    PGN_AFTERTREATMENT_1_GAS_OXIDATION_CATALYST : UDINT := UDINT#16#FD22; (* < 64802 - A1GOC *)
    PGN_EXTENDED_JOYSTICK_MESSAGE_10 : UDINT := UDINT#16#FD23; (* < 64803 - EJM10 *)
    PGN_BASIC_JOYSTICK_MESSAGE_10 : UDINT := UDINT#16#FD24; (* < 64804 - BJM10 *)
    PGN_EXTENDED_JOYSTICK_MESSAGE_9 : UDINT := UDINT#16#FD25; (* < 64805 - EJM9 *)
    PGN_BASIC_JOYSTICK_MESSAGE_9 : UDINT := UDINT#16#FD26; (* < 64806 - BJM9 *)
    PGN_EXTENDED_JOYSTICK_MESSAGE_8 : UDINT := UDINT#16#FD27; (* < 64807 - EJM8 *)
    PGN_BASIC_JOYSTICK_MESSAGE_8 : UDINT := UDINT#16#FD28; (* < 64808 - BJM8 *)
    PGN_EXTENDED_JOYSTICK_MESSAGE_7 : UDINT := UDINT#16#FD29; (* < 64809 - EJM7 *)
    PGN_BASIC_JOYSTICK_MESSAGE_7 : UDINT := UDINT#16#FD2A; (* < 64810 - BJM7 *)
    PGN_EXTENDED_JOYSTICK_MESSAGE_6 : UDINT := UDINT#16#FD2B; (* < 64811 - EJM6 *)
    PGN_BASIC_JOYSTICK_MESSAGE_6 : UDINT := UDINT#16#FD2C; (* < 64812 - BJM6 *)
    PGN_EXTENDED_JOYSTICK_MESSAGE_5 : UDINT := UDINT#16#FD2D; (* < 64813 - EJM5 *)
    PGN_BASIC_JOYSTICK_MESSAGE_5 : UDINT := UDINT#16#FD2E; (* < 64814 - BJM5 *)
    PGN_EXTENDED_JOYSTICK_MESSAGE_4 : UDINT := UDINT#16#FD2F; (* < 64815 - EJM4 *)
    PGN_BASIC_JOYSTICK_MESSAGE_4 : UDINT := UDINT#16#FD30; (* < 64816 - BJM4 *)
    PGN_FAN_DRIVE_2 : UDINT := UDINT#16#FD31; (* < 64817 - FD2 *)
    PGN_ECU_DIAGNOSTIC_PROTOCOL : UDINT := UDINT#16#FD32; (* < 64818 - ECUDP *)
    PGN_AFTERTREATMENT_2_DIESEL_EXHAUST_FLUID_SUPPLY_INFORMATION : UDINT := UDINT#16#FD33; (* < 64819 - A2DEFSI *)
    PGN_AFTERTREATMENT_2_SCR_REAGANT_TANK_2_INFORMATION : UDINT := UDINT#16#FD34; (* < 64820 - A2SCRRT2I *)
    PGN_AFTERTREATMENT_2_DIESEL_EXHAUST_FLUID_TANK_1_INFORMATION_1 : UDINT := UDINT#16#FD35; (* < 64821 - A2DEFT1I1 *)
    PGN_AFTERTREATMENT_2_DIESEL_EXHAUST_FLUID_INFORMATION_1 : UDINT := UDINT#16#FD36; (* < 64822 - A2DEFI1 *)
    PGN_AFTERTREATMENT_2_SCR_SERVICE_INFORMATION_1 : UDINT := UDINT#16#FD37; (* < 64823 - A2SCRSI1 *)
    PGN_AFTERTREATMENT_2_SCR_EXHAUST_GAS_TEMPERATURE_1 : UDINT := UDINT#16#FD38; (* < 64824 - A2SCREGT1 *)
    PGN_AFTERTREATMENT_2_SCR_EXHAUST_GAS_PRESSURES : UDINT := UDINT#16#FD39; (* < 64825 - A2SCREGP *)
    PGN_AFTERTREATMENT_2_SCR_DOSING_SYSTEM_REQUESTS_2 : UDINT := UDINT#16#FD3A; (* < 64826 - A2SCRDSR2 *)
    PGN_AFTERTREATMENT_2_SCR_DOSING_SYSTEM_INFORMATION_2 : UDINT := UDINT#16#FD3B; (* < 64827 - A2SCRDSI2 *)
    PGN_AFTERTREATMENT_1_DIESEL_EXHAUST_FLUID_SUPPLY_INFORMATION : UDINT := UDINT#16#FD3C; (* < 64828 - A1DEFSI *)
    PGN_AFTERTREATMENT_1_SCR_REAGANT_TANK_2_INFORMATION : UDINT := UDINT#16#FD3D; (* < 64829 - A1SCRRT2I *)
    PGN_AFTERTREATMENT_1_SCR_EXHAUST_GAS_TEMPERATURE_1 : UDINT := UDINT#16#FD3E; (* < 64830 - A1SCREGT1 *)
    PGN_AFTERTREATMENT_1_SCR_EXHAUST_GAS_PRESSURES : UDINT := UDINT#16#FD3F; (* < 64831 - A1SCREGP *)
    PGN_AFTERTREATMENT_1_SCR_DOSING_SYSTEM_REQUESTS_2 : UDINT := UDINT#16#FD40; (* < 64832 - A1SCRDSR2 *)
    PGN_AFTERTREATMENT_1_SCR_DOSING_SYSTEM_INFORMATION_2 : UDINT := UDINT#16#FD41; (* < 64833 - A1SCRDSI2 *)
    PGN_ISOBUS_COMPLIANCE_CERTIFICA : UDINT := UDINT#16#FD42; (* < 64834 - ICC *)
    PGN_MACHINE_SELECT_SPEED_CMD : UDINT := UDINT#16#FD43; (* < 64835 - MSSC *)
